   DATA[2664,36] := 1.730048;
   DATA[2664,37] := 188.8618;
   DATA[2664,38] := 0.000128152;
   DATA[2664,39] := 1.0;
   DATA[2664,40] := 1.0;
   DATA[2665,0] := 2.431861;
   DATA[2665,1] := 870.5869;
   DATA[2665,2] := 2.0;
   DATA[2665,3] := 2.0;
   DATA[2665,4] := 262.3366;
   DATA[2665,5] := 8.396757;
   DATA[2665,6] := 329.1464;
   DATA[2665,7] := 2.451799;
   DATA[2665,8] := 2.0;
   DATA[2665,9] := 2.0;
   DATA[2665,10] := 2.0;
   DATA[2665,11] := 19.69396;
   DATA[2665,12] := 2.206322;
   DATA[2665,13] := 834.4415;
   DATA[2665,14] := 1.0;
   DATA[2665,15] := 2.0;
   DATA[2665,16] := 1.0;
   DATA[2665,17] := 1.0;
   DATA[2665,18] := 1.0;
   DATA[2665,19] := 2.0;
   DATA[2665,20] := 148.808;
   DATA[2665,21] := 155.3961;
   DATA[2665,22] := 1.717233;
   DATA[2665,23] := 881.2356;
   DATA[2665,24] := 2.0;
   DATA[2665,25] := 2.0;
   DATA[2665,26] := 7.872853;
   DATA[2665,27] := 144.7065;
   DATA[2665,28] := 261.3432;
   DATA[2665,29] := 12.03538;
   DATA[2665,30] := 1.726352;
   DATA[2665,31] := 1.3119;
   DATA[2665,32] := 0.7352687;
   DATA[2665,33] := 0.3066329;
   DATA[2665,34] := 2.0;
   DATA[2665,35] := 250.0961;
   DATA[2665,36] := 1.730048;
   DATA[2665,37] := 188.8618;
   DATA[2665,38] := 0.000128152;
   DATA[2665,39] := 1.0;
   DATA[2665,40] := 1.0;
   DATA[2666,0] := 2.431861;
   DATA[2666,1] := 870.4692;
   DATA[2666,2] := 2.0;
   DATA[2666,3] := 2.0;
   DATA[2666,4] := 262.3366;
   DATA[2666,5] := 8.396757;
   DATA[2666,6] := 329.1464;
   DATA[2666,7] := 2.451799;
   DATA[2666,8] := 2.0;
   DATA[2666,9] := 2.0;
   DATA[2666,10] := 2.0;
   DATA[2666,11] := 19.72598;
   DATA[2666,12] := 2.206322;
   DATA[2666,13] := 834.4415;
   DATA[2666,14] := 1.0;
   DATA[2666,15] := 2.0;
   DATA[2666,16] := 1.0;
   DATA[2666,17] := 1.0;
   DATA[2666,18] := 1.0;
   DATA[2666,19] := 2.0;
   DATA[2666,20] := 148.808;
   DATA[2666,21] := 155.3961;
   DATA[2666,22] := 1.717233;
   DATA[2666,23] := 881.4663;
   DATA[2666,24] := 2.0;
   DATA[2666,25] := 2.0;
   DATA[2666,26] := 7.872853;
   DATA[2666,27] := 144.7065;
   DATA[2666,28] := 261.3432;
   DATA[2666,29] := 12.03538;
   DATA[2666,30] := 1.726352;
   DATA[2666,31] := 1.30652;
   DATA[2666,32] := 0.7352687;
   DATA[2666,33] := 0.3066329;
   DATA[2666,34] := 2.0;
   DATA[2666,35] := 250.0961;
   DATA[2666,36] := 1.730048;
   DATA[2666,37] := 188.8618;
   DATA[2666,38] := 0.000128152;
   DATA[2666,39] := 1.0;
   DATA[2666,40] := 1.0;
   DATA[2667,0] := 2.455882;
   DATA[2667,1] := 870.5869;
   DATA[2667,2] := 2.0;
   DATA[2667,3] := 2.0;
   DATA[2667,4] := 262.3366;
   DATA[2667,5] := 8.396757;
   DATA[2667,6] := 329.1464;
   DATA[2667,7] := 2.455131;
   DATA[2667,8] := 2.0;
   DATA[2667,9] := 2.0;
   DATA[2667,10] := 2.0;
   DATA[2667,11] := 19.74198;
   DATA[2667,12] := 2.20645;
   DATA[2667,13] := 834.802;
   DATA[2667,14] := 1.0;
   DATA[2667,15] := 2.0;
   DATA[2667,16] := 1.0;
   DATA[2667,17] := 1.0;
   DATA[2667,18] := 1.0;
   DATA[2667,19] := 2.0;
   DATA[2667,20] := 148.808;
   DATA[2667,21] := 155.3961;
   DATA[2667,22] := 1.719156;
   DATA[2667,23] := 882.0431;
   DATA[2667,24] := 2.0;
   DATA[2667,25] := 2.0;
   DATA[2667,26] := 7.872853;
   DATA[2667,27] := 144.7065;
   DATA[2667,28] := 261.3432;
   DATA[2667,29] := 12.03538;
   DATA[2667,30] := 1.726352;
   DATA[2667,31] := 1.311387;
   DATA[2667,32] := 0.7352687;
   DATA[2667,33] := 0.3066329;
   DATA[2667,34] := 2.0;
   DATA[2667,35] := 250.1442;
   DATA[2667,36] := 1.730048;
   DATA[2667,37] := 188.8618;
   DATA[2667,38] := 0.000128152;
   DATA[2667,39] := 1.0;
   DATA[2667,40] := 1.0;
   DATA[2668,0] := 2.50008;
   DATA[2668,1] := 870.3907;
   DATA[2668,2] := 2.0;
   DATA[2668,3] := 2.0;
   DATA[2668,4] := 262.3366;
   DATA[2668,5] := 8.396757;
   DATA[2668,6] := 329.1464;
   DATA[2668,7] := 2.455131;
   DATA[2668,8] := 2.0;
   DATA[2668,9] := 2.0;
   DATA[2668,10] := 2.0;
   DATA[2668,11] := 19.75799;
   DATA[2668,12] := 2.209909;
   DATA[2668,13] := 834.802;
   DATA[2668,14] := 1.0;
   DATA[2668,15] := 2.0;
   DATA[2668,16] := 1.0;
   DATA[2668,17] := 1.0;
   DATA[2668,18] := 1.0;
   DATA[2668,19] := 2.0;
   DATA[2668,20] := 148.808;
   DATA[2668,21] := 155.3961;
   DATA[2668,22] := 1.719156;
   DATA[2668,23] := 882.1969;
   DATA[2668,24] := 2.0;
   DATA[2668,25] := 2.0;
   DATA[2668,26] := 7.872853;
   DATA[2668,27] := 144.7065;
   DATA[2668,28] := 261.3432;
   DATA[2668,29] := 12.03538;
   DATA[2668,30] := 1.726352;
   DATA[2668,31] := 1.313949;
   DATA[2668,32] := 0.7352687;
   DATA[2668,33] := 0.3066329;
   DATA[2668,34] := 2.0;
   DATA[2668,35] := 250.3044;
   DATA[2668,36] := 1.730048;
   DATA[2668,37] := 189.0381;
   DATA[2668,38] := 0.000128152;
   DATA[2668,39] := 1.0;
   DATA[2668,40] := 1.0;
   DATA[2669,0] := 2.537873;
   DATA[2669,1] := 870.7047;
   DATA[2669,2] := 2.0;
   DATA[2669,3] := 2.0;
   DATA[2669,4] := 262.3366;
   DATA[2669,5] := 8.396757;
   DATA[2669,6] := 329.1464;
   DATA[2669,7] := 2.455131;
   DATA[2669,8] := 2.0;
   DATA[2669,9] := 2.0;
   DATA[2669,10] := 2.0;
   DATA[2669,11] := 19.7964;
   DATA[2669,12] := 2.209909;
   DATA[2669,13] := 835.1625;
   DATA[2669,14] := 1.0;
   DATA[2669,15] := 2.0;
   DATA[2669,16] := 1.0;
   DATA[2669,17] := 1.0;
   DATA[2669,18] := 1.0;
   DATA[2669,19] := 2.0;
   DATA[2669,20] := 148.808;
   DATA[2669,21] := 155.3961;
   DATA[2669,22] := 1.719156;
   DATA[2669,23] := 882.2354;
   DATA[2669,24] := 2.0;
   DATA[2669,25] := 2.0;
   DATA[2669,26] := 7.874135;
   DATA[2669,27] := 144.7065;
   DATA[2669,28] := 261.3432;
   DATA[2669,29] := 12.03538;
   DATA[2669,30] := 1.726352;
   DATA[2669,31] := 1.311643;
   DATA[2669,32] := 0.7352687;
   DATA[2669,33] := 0.3066329;
   DATA[2669,34] := 2.0;
   DATA[2669,35] := 250.3044;
   DATA[2669,36] := 1.730048;
   DATA[2669,37] := 189.0541;
   DATA[2669,38] := 0.000128152;
   DATA[2669,39] := 1.0;
   DATA[2669,40] := 1.0;
   DATA[2670,0] := 2.585594;
   DATA[2670,1] := 871.058;
   DATA[2670,2] := 2.0;
   DATA[2670,3] := 2.0;
   DATA[2670,4] := 262.3366;
   DATA[2670,5] := 8.396757;
   DATA[2670,6] := 329.1464;
   DATA[2670,7] := 2.455131;
   DATA[2670,8] := 2.0;
   DATA[2670,9] := 2.0;
   DATA[2670,10] := 2.0;
   DATA[2670,11] := 19.7964;
   DATA[2670,12] := 2.209909;
   DATA[2670,13] := 835.1625;
   DATA[2670,14] := 1.0;
   DATA[2670,15] := 2.0;
   DATA[2670,16] := 1.0;
   DATA[2670,17] := 1.0;
   DATA[2670,18] := 1.0;
   DATA[2670,19] := 2.0;
   DATA[2670,20] := 148.808;
   DATA[2670,21] := 155.3961;
   DATA[2670,22] := 1.717105;
   DATA[2670,23] := 882.3892;
   DATA[2670,24] := 2.0;
   DATA[2670,25] := 2.0;
   DATA[2670,26] := 7.874135;
   DATA[2670,27] := 144.7065;
   DATA[2670,28] := 261.3432;
   DATA[2670,29] := 12.03538;
   DATA[2670,30] := 1.726352;
   DATA[2670,31] := 1.288587;
   DATA[2670,32] := 0.7352687;
   DATA[2670,33] := 0.3066329;
   DATA[2670,34] := 2.0;
   DATA[2670,35] := 250.3044;
   DATA[2670,36] := 1.730048;
   DATA[2670,37] := 189.1182;
   DATA[2670,38] := 0.000128152;
   DATA[2670,39] := 1.0;
   DATA[2670,40] := 1.0;
   DATA[2671,0] := 2.618903;
   DATA[2671,1] := 870.7047;
   DATA[2671,2] := 2.0;
   DATA[2671,3] := 2.0;
   DATA[2671,4] := 262.3366;
   DATA[2671,5] := 8.396757;
   DATA[2671,6] := 329.1464;
   DATA[2671,7] := 2.456156;
   DATA[2671,8] := 2.0;
   DATA[2671,9] := 2.0;
   DATA[2671,10] := 2.0;
   DATA[2671,11] := 19.7804;
   DATA[2671,12] := 2.209909;
   DATA[2671,13] := 835.2025;
   DATA[2671,14] := 1.0;
   DATA[2671,15] := 2.0;
   DATA[2671,16] := 1.0;
   DATA[2671,17] := 1.0;
   DATA[2671,18] := 1.0;
   DATA[2671,19] := 2.0;
   DATA[2671,20] := 148.808;
   DATA[2671,21] := 155.3961;
   DATA[2671,22] := 1.717105;
   DATA[2671,23] := 882.6967;
   DATA[2671,24] := 2.0;
   DATA[2671,25] := 2.0;
   DATA[2671,26] := 7.874135;
   DATA[2671,27] := 144.7065;
   DATA[2671,28] := 261.3432;
   DATA[2671,29] := 12.03538;
   DATA[2671,30] := 1.726352;
   DATA[2671,31] := 1.27296;
   DATA[2671,32] := 0.7352687;
   DATA[2671,33] := 0.3066329;
   DATA[2671,34] := 2.0;
   DATA[2671,35] := 250.3044;
   DATA[2671,36] := 1.730048;
   DATA[2671,37] := 189.1182;
   DATA[2671,38] := 0.000128152;
   DATA[2671,39] := 1.0;
   DATA[2671,40] := 1.0;
   DATA[2672,0] := 2.644845;
   DATA[2672,1] := 871.2542;
   DATA[2672,2] := 2.0;
   DATA[2672,3] := 2.0;
   DATA[2672,4] := 262.3366;
   DATA[2672,5] := 8.396757;
   DATA[2672,6] := 329.1464;
   DATA[2672,7] := 2.456156;
   DATA[2672,8] := 2.0;
   DATA[2672,9] := 2.0;
   DATA[2672,10] := 2.0;
   DATA[2672,11] := 19.73558;
   DATA[2672,12] := 2.209909;
   DATA[2672,13] := 835.2827;
   DATA[2672,14] := 1.0;
   DATA[2672,15] := 2.0;
   DATA[2672,16] := 1.0;
   DATA[2672,17] := 1.0;
   DATA[2672,18] := 1.0;
   DATA[2672,19] := 2.0;
   DATA[2672,20] := 148.808;
   DATA[2672,21] := 155.3961;
   DATA[2672,22] := 1.717105;
   DATA[2672,23] := 882.8121;
   DATA[2672,24] := 2.0;
   DATA[2672,25] := 2.0;
   DATA[2672,26] := 7.874135;
   DATA[2672,27] := 144.7065;
   DATA[2672,28] := 261.3432;
   DATA[2672,29] := 12.03538;
   DATA[2672,30] := 1.726352;
   DATA[2672,31] := 1.265915;
   DATA[2672,32] := 0.7352687;
   DATA[2672,33] := 0.3066329;
   DATA[2672,34] := 2.0;
   DATA[2672,35] := 250.3044;
   DATA[2672,36] := 1.730048;
   DATA[2672,37] := 188.9419;
   DATA[2672,38] := 0.000128152;
   DATA[2672,39] := 1.0;
   DATA[2672,40] := 1.0;
   DATA[2673,0] := 2.658937;
   DATA[2673,1] := 871.058;
   DATA[2673,3] := 2.0;
   DATA[2673,4] := 262.3366;
   DATA[2673,5] := 8.396757;
   DATA[2673,6] := 329.1464;
   DATA[2673,7] := 2.456156;
   DATA[2673,8] := 2.0;
   DATA[2673,9] := 2.0;
   DATA[2673,10] := 2.0;
   DATA[2673,11] := 19.71637;
   DATA[2673,12] := 2.211959;
   DATA[2673,13] := 835.6832;
   DATA[2673,14] := 1.0;
   DATA[2673,15] := 2.0;
   DATA[2673,16] := 1.0;
   DATA[2673,17] := 1.0;
   DATA[2673,18] := 1.0;
   DATA[2673,19] := 2.0;
   DATA[2673,20] := 148.808;
   DATA[2673,21] := 155.3961;
   DATA[2673,22] := 1.717105;
   DATA[2673,23] := 882.6967;
   DATA[2673,24] := 2.0;
   DATA[2673,25] := 2.0;
   DATA[2673,26] := 7.874135;
   DATA[2673,27] := 144.7065;
   DATA[2673,28] := 261.3432;
   DATA[2673,29] := 12.03538;
   DATA[2673,30] := 1.728659;
   DATA[2673,31] := 1.261944;
   DATA[2673,32] := 0.7352687;
   DATA[2673,33] := 0.3066329;
   DATA[2673,34] := 2.0;
   DATA[2673,35] := 250.3044;
   DATA[2673,36] := 1.730048;
   DATA[2673,37] := 188.9419;
   DATA[2673,38] := 0.000128152;
   DATA[2673,39] := 1.0;
   DATA[2673,40] := 1.0;
   DATA[2674,0] := 2.658937;
   DATA[2674,1] := 871.0972;
   DATA[2674,3] := 2.0;
   DATA[2674,4] := 262.3366;
   DATA[2674,5] := 8.396757;
   DATA[2674,6] := 329.1464;
   DATA[2674,7] := 2.453978;
   DATA[2674,8] := 2.0;
   DATA[2674,9] := 2.0;
   DATA[2674,10] := 2.0;
   DATA[2674,11] := 19.71637;
   DATA[2674,12] := 2.212215;
   DATA[2674,13] := 835.563;
   DATA[2674,14] := 1.0;
   DATA[2674,15] := 2.0;
   DATA[2674,16] := 1.0;
   DATA[2674,17] := 1.0;
   DATA[2674,18] := 1.0;
   DATA[2674,19] := 2.0;
   DATA[2674,20] := 148.808;
   DATA[2674,21] := 155.3961;
   DATA[2674,22] := 1.717105;
   DATA[2674,23] := 882.889;
   DATA[2674,24] := 2.0;
   DATA[2674,25] := 2.0;
   DATA[2674,26] := 7.874135;
   DATA[2674,27] := 144.7065;
   DATA[2674,28] := 261.3432;
   DATA[2674,29] := 12.03538;
   DATA[2674,30] := 1.728916;
   DATA[2674,31] := 1.276419;
   DATA[2674,32] := 0.7352687;
   DATA[2674,33] := 0.3066329;
   DATA[2674,34] := 2.0;
   DATA[2674,35] := 250.1442;
   DATA[2674,36] := 1.730048;
   DATA[2674,37] := 188.9419;
   DATA[2674,38] := 0.000128152;
   DATA[2674,39] := 1.0;
   DATA[2674,40] := 1.0;
   DATA[2675,0] := 2.639721;
   DATA[2675,1] := 871.215;
   DATA[2675,3] := 2.0;
   DATA[2675,4] := 262.3366;
   DATA[2675,5] := 8.396757;
   DATA[2675,6] := 329.1464;
   DATA[2675,7] := 2.452952;
   DATA[2675,8] := 2.0;
   DATA[2675,9] := 2.0;
   DATA[2675,10] := 2.0;
   DATA[2675,11] := 19.71637;
   DATA[2675,12] := 2.212215;
   DATA[2675,13] := 835.4028;
   DATA[2675,14] := 1.0;
   DATA[2675,15] := 2.0;
   DATA[2675,16] := 1.0;
   DATA[2675,17] := 1.0;
   DATA[2675,18] := 1.0;
   DATA[2675,19] := 2.0;
   DATA[2675,20] := 148.808;
   DATA[2675,21] := 155.3961;
   DATA[2675,22] := 1.717105;
   DATA[2675,23] := 882.6198;
   DATA[2675,24] := 2.0;
   DATA[2675,25] := 2.0;
   DATA[2675,26] := 7.874135;
   DATA[2675,27] := 144.7065;
   DATA[2675,28] := 261.3432;
   DATA[2675,29] := 11.72776;
   DATA[2675,30] := 1.728916;
   DATA[2675,31] := 1.28167;
   DATA[2675,32] := 0.7352687;
   DATA[2675,33] := 0.3066329;
   DATA[2675,34] := 2.0;
   DATA[2675,35] := 250.1442;
   DATA[2675,36] := 1.730048;
   DATA[2675,37] := 188.9419;
   DATA[2675,38] := 0.000128152;
   DATA[2675,39] := 1.0;
   DATA[2675,40] := 1.0;
   DATA[2676,0] := 2.633635;
   DATA[2676,1] := 870.9794;
   DATA[2676,3] := 2.0;
   DATA[2676,4] := 262.3366;
   DATA[2676,5] := 8.396757;
   DATA[2676,6] := 329.1464;
   DATA[2676,7] := 2.452952;
   DATA[2676,8] := 2.0;
   DATA[2676,9] := 2.0;
   DATA[2676,10] := 2.0;
   DATA[2676,11] := 19.71637;
   DATA[2676,12] := 2.209397;
   DATA[2676,13] := 835.6031;
   DATA[2676,14] := 1.0;
   DATA[2676,15] := 2.0;
   DATA[2676,16] := 1.0;
   DATA[2676,17] := 1.0;
   DATA[2676,18] := 1.0;
   DATA[2676,19] := 2.0;
   DATA[2676,20] := 148.808;
   DATA[2676,21] := 155.5242;
   DATA[2676,22] := 1.717105;
   DATA[2676,23] := 882.5814;
   DATA[2676,24] := 2.0;
   DATA[2676,25] := 2.0;
   DATA[2676,26] := 7.874135;
   DATA[2676,27] := 144.7065;
   DATA[2676,28] := 261.3432;
   DATA[2676,29] := 11.72776;
   DATA[2676,30] := 1.728916;
   DATA[2676,31] := 1.276547;
   DATA[2676,32] := 0.7352687;
   DATA[2676,33] := 0.3066329;
   DATA[2676,34] := 2.0;
   DATA[2676,35] := 250.3525;
   DATA[2676,36] := 1.730048;
   DATA[2676,37] := 189.1182;
   DATA[2676,38] := 0.000128152;
   DATA[2676,39] := 1.0;
   DATA[2676,40] := 1.0;
   DATA[2677,0] := 2.633635;
   DATA[2677,1] := 870.6654;
   DATA[2677,3] := 2.0;
   DATA[2677,4] := 262.3366;
   DATA[2677,5] := 8.396757;
   DATA[2677,6] := 329.1464;
   DATA[2677,7] := 2.452952;
   DATA[2677,8] := 2.0;
   DATA[2677,9] := 2.0;
   DATA[2677,10] := 2.0;
   DATA[2677,11] := 19.71637;
   DATA[2677,12] := 2.209397;
   DATA[2677,13] := 835.4429;
   DATA[2677,14] := 1.0;
   DATA[2677,15] := 2.0;
   DATA[2677,16] := 1.0;
   DATA[2677,17] := 1.0;
   DATA[2677,18] := 1.0;
   DATA[2677,19] := 2.0;
   DATA[2677,20] := 148.808;
   DATA[2677,21] := 155.5242;
   DATA[2677,22] := 1.718515;
   DATA[2677,23] := 882.6967;
   DATA[2677,24] := 2.0;
   DATA[2677,25] := 2.0;
   DATA[2677,26] := 7.874135;
   DATA[2677,27] := 144.7065;
   DATA[2677,28] := 261.3432;
   DATA[2677,29] := 11.72776;
   DATA[2677,30] := 1.730838;
   DATA[2677,31] := 1.280902;
   DATA[2677,32] := 0.7352687;
   DATA[2677,33] := 0.3084905;
   DATA[2677,34] := 2.0;
   DATA[2677,35] := 250.3525;
   DATA[2677,36] := 1.730048;
   DATA[2677,37] := 189.1182;
   DATA[2677,38] := 0.000128152;
   DATA[2677,39] := 1.0;
   DATA[2677,40] := 1.0;
   DATA[2678,0] := 2.625628;
   DATA[2678,1] := 870.6654;
   DATA[2678,3] := 2.0;
   DATA[2678,4] := 262.3366;
   DATA[2678,5] := 8.396757;
   DATA[2678,6] := 329.1464;
   DATA[2678,7] := 2.452952;
   DATA[2678,8] := 2.0;
   DATA[2678,9] := 2.0;
   DATA[2678,10] := 2.0;
   DATA[2678,11] := 19.73878;
   DATA[2678,12] := 2.209397;
   DATA[2678,13] := 835.3627;
   DATA[2678,14] := 1.0;
   DATA[2678,15] := 2.0;
   DATA[2678,16] := 1.0;
   DATA[2678,17] := 1.0;
   DATA[2678,18] := 1.0;
   DATA[2678,19] := 2.0;
   DATA[2678,20] := 148.808;
   DATA[2678,21] := 155.5242;
   DATA[2678,22] := 1.718515;
   DATA[2678,23] := 882.6583;
   DATA[2678,24] := 2.0;
   DATA[2678,25] := 2.0;
   DATA[2678,26] := 7.874135;
   DATA[2678,27] := 144.7065;
   DATA[2678,28] := 261.3432;
   DATA[2678,29] := 12.07383;
   DATA[2678,30] := 1.731735;
   DATA[2678,31] := 1.288203;
   DATA[2678,32] := 0.7352687;
   DATA[2678,33] := 0.3084905;
   DATA[2678,34] := 2.0;
   DATA[2678,35] := 250.4967;
   DATA[2678,36] := 1.730048;
   DATA[2678,37] := 189.2624;
   DATA[2678,38] := 0.000128152;
   DATA[2678,39] := 1.0;
   DATA[2678,40] := 1.0;
   DATA[2679,0] := 2.600006;
   DATA[2679,1] := 871.058;
   DATA[2679,3] := 2.0;
   DATA[2679,4] := 262.3366;
   DATA[2679,5] := 8.396757;
   DATA[2679,6] := 329.1464;
   DATA[2679,7] := 2.452952;
   DATA[2679,8] := 2.0;
   DATA[2679,9] := 2.0;
   DATA[2679,10] := 2.0;
   DATA[2679,11] := 19.74838;
   DATA[2679,12] := 2.209397;
   DATA[2679,13] := 835.0023;
   DATA[2679,14] := 1.0;
   DATA[2679,15] := 2.0;
   DATA[2679,16] := 1.0;
   DATA[2679,17] := 1.0;
   DATA[2679,18] := 1.0;
   DATA[2679,19] := 2.0;
   DATA[2679,20] := 148.808;
   DATA[2679,21] := 155.473;
   DATA[2679,22] := 1.718515;
   DATA[2679,23] := 882.4661;
   DATA[2679,24] := 2.0;
   DATA[2679,25] := 2.0;
   DATA[2679,26] := 7.874135;
   DATA[2679,27] := 144.7065;
   DATA[2679,28] := 261.3432;
   DATA[2679,29] := 12.07383;
   DATA[2679,30] := 1.731735;
   DATA[2679,31] := 1.307416;
   DATA[2679,32] := 0.7352687;
   DATA[2679,33] := 0.3084905;
   DATA[2679,34] := 2.0;
   DATA[2679,35] := 250.4967;
   DATA[2679,36] := 1.730048;
   DATA[2679,37] := 189.2624;
   DATA[2679,38] := 0.000128152;
   DATA[2679,39] := 1.0;
   DATA[2679,40] := 1.0;
   DATA[2680,0] := 2.552285;
   DATA[2680,1] := 870.7047;
   DATA[2680,3] := 2.0;
   DATA[2680,4] := 262.3366;
   DATA[2680,5] := 8.396757;
   DATA[2680,6] := 329.0182;
   DATA[2680,7] := 2.452568;
   DATA[2680,8] := 2.0;
   DATA[2680,9] := 2.0;
   DATA[2680,10] := 2.0;
   DATA[2680,11] := 19.74838;
   DATA[2680,12] := 2.20645;
   DATA[2680,13] := 834.762;
   DATA[2680,14] := 1.0;
   DATA[2680,15] := 2.0;
   DATA[2680,16] := 1.0;
   DATA[2680,17] := 1.0;
   DATA[2680,18] := 1.0;
   DATA[2680,19] := 2.0;
   DATA[2680,20] := 148.808;
   DATA[2680,21] := 155.4473;
   DATA[2680,22] := 1.718515;
   DATA[2680,23] := 882.5045;
   DATA[2680,24] := 2.0;
   DATA[2680,25] := 2.0;
   DATA[2680,26] := 7.870931;
   DATA[2680,27] := 144.7834;
   DATA[2680,28] := 261.3432;
   DATA[2680,29] := 12.07383;
   DATA[2680,30] := 1.731735;
   DATA[2680,31] := 1.320994;
   DATA[2680,32] := 0.7352687;
   DATA[2680,33] := 0.3084905;
   DATA[2680,34] := 2.0;
   DATA[2680,35] := 250.4967;
   DATA[2680,36] := 1.730048;
   DATA[2680,37] := 189.2624;
   DATA[2680,38] := 0.000128152;
   DATA[2680,39] := 1.0;
   DATA[2680,40] := 1.0;
   DATA[2681,0] := 2.499119;
   DATA[2681,1] := 870.8224;
   DATA[2681,3] := 2.0;
   DATA[2681,4] := 262.3366;
   DATA[2681,5] := 8.396757;
   DATA[2681,6] := 329.0182;
   DATA[2681,7] := 2.451671;
   DATA[2681,8] := 2.0;
   DATA[2681,9] := 2.0;
   DATA[2681,10] := 2.0;
   DATA[2681,11] := 19.74838;
   DATA[2681,12] := 2.20645;
   DATA[2681,13] := 834.6818;
   DATA[2681,14] := 1.0;
   DATA[2681,15] := 2.0;
   DATA[2681,16] := 1.0;
   DATA[2681,17] := 1.0;
   DATA[2681,18] := 1.0;
   DATA[2681,19] := 2.0;
   DATA[2681,20] := 148.808;
   DATA[2681,21] := 155.4473;
   DATA[2681,22] := 1.718515;
   DATA[2681,23] := 882.12;
   DATA[2681,24] := 2.0;
   DATA[2681,25] := 2.0;
   DATA[2681,26] := 7.870931;
   DATA[2681,27] := 144.7834;
   DATA[2681,28] := 261.3432;
   DATA[2681,29] := 12.07383;
   DATA[2681,30] := 1.731735;
   DATA[2681,31] := 1.329064;
   DATA[2681,32] := 0.7352687;
   DATA[2681,33] := 0.3084905;
   DATA[2681,34] := 2.0;
   DATA[2681,35] := 250.4967;
   DATA[2681,36] := 1.730048;
   DATA[2681,37] := 189.2624;
   DATA[2681,38] := 0.000128152;
   DATA[2681,39] := 1.0;
   DATA[2681,40] := 1.0;
   DATA[2682,0] := 2.400154;
   DATA[2682,1] := 870.6654;
   DATA[2682,2] := 1.0;
   DATA[2682,3] := 2.0;
   DATA[2682,4] := 262.3366;
   DATA[2682,5] := 8.396757;
   DATA[2682,6] := 329.0182;
   DATA[2682,7] := 2.451671;
   DATA[2682,8] := 2.0;
   DATA[2682,9] := 2.0;
   DATA[2682,10] := 2.0;
   DATA[2682,11] := 19.74838;
   DATA[2682,12] := 2.20645;
   DATA[2682,13] := 835.2025;
   DATA[2682,14] := 1.0;
   DATA[2682,15] := 2.0;
   DATA[2682,16] := 1.0;
   DATA[2682,17] := 1.0;
   DATA[2682,18] := 1.0;
   DATA[2682,19] := 2.0;
   DATA[2682,20] := 148.808;
   DATA[2682,21] := 155.4473;
   DATA[2682,22] := 1.718515;
   DATA[2682,23] := 882.2738;
   DATA[2682,24] := 2.0;
   DATA[2682,25] := 2.0;
   DATA[2682,26] := 7.873815;
   DATA[2682,27] := 144.7834;
   DATA[2682,28] := 261.3432;
   DATA[2682,29] := 12.07383;
   DATA[2682,30] := 1.731351;
   DATA[2682,31] := 1.332138;
   DATA[2682,32] := 0.7352687;
   DATA[2682,33] := 0.3084905;
   DATA[2682,34] := 2.0;
   DATA[2682,35] := 250.4967;
   DATA[2682,36] := 1.730048;
   DATA[2682,37] := 189.2624;
   DATA[2682,38] := 0.000128152;
   DATA[2682,39] := 1.0;
   DATA[2682,40] := 1.0;
   DATA[2683,0] := 2.223361;
   DATA[2683,1] := 870.9794;
   DATA[2683,2] := 1.0;
   DATA[2683,3] := 2.0;
   DATA[2683,4] := 262.3366;
   DATA[2683,5] := 8.396757;
   DATA[2683,6] := 329.0182;
   DATA[2683,7] := 2.451671;
   DATA[2683,8] := 2.0;
   DATA[2683,9] := 2.0;
   DATA[2683,10] := 2.0;
   DATA[2683,11] := 19.74838;
   DATA[2683,12] := 2.20645;
   DATA[2683,13] := 834.6818;
   DATA[2683,14] := 1.0;
   DATA[2683,15] := 2.0;
   DATA[2683,16] := 1.0;
   DATA[2683,17] := 1.0;
   DATA[2683,18] := 1.0;
   DATA[2683,19] := 2.0;
   DATA[2683,20] := 148.808;
   DATA[2683,21] := 155.4473;
   DATA[2683,22] := 1.718515;
   DATA[2683,23] := 882.5045;
   DATA[2683,24] := 2.0;
   DATA[2683,25] := 2.0;
   DATA[2683,26] := 7.874776;
   DATA[2683,27] := 144.7834;
   DATA[2683,28] := 261.3432;
   DATA[2683,29] := 12.07383;
   DATA[2683,30] := 1.731351;
   DATA[2683,31] := 1.31523;
   DATA[2683,32] := 0.7352687;
   DATA[2683,33] := 0.3084905;
   DATA[2683,34] := 2.0;
   DATA[2683,35] := 250.4967;
   DATA[2683,36] := 1.810143;
   DATA[2683,37] := 189.2624;
   DATA[2683,38] := 0.000128152;
   DATA[2683,39] := 1.0;
   DATA[2683,40] := 1.0;
   DATA[2684,0] := 1.916216;
   DATA[2684,1] := 870.5869;
   DATA[2684,2] := 1.0;
   DATA[2684,3] := 2.0;
   DATA[2684,4] := 262.3366;
   DATA[2684,5] := 8.396757;
   DATA[2684,6] := 329.0182;
   DATA[2684,7] := 2.451671;
   DATA[2684,8] := 2.0;
   DATA[2684,9] := 2.0;
   DATA[2684,10] := 2.0;
   DATA[2684,11] := 19.74838;
   DATA[2684,12] := 2.207091;
   DATA[2684,13] := 835.2025;
   DATA[2684,14] := 1.0;
   DATA[2684,15] := 2.0;
   DATA[2684,16] := 1.0;
   DATA[2684,17] := 1.0;
   DATA[2684,18] := 1.0;
   DATA[2684,19] := 2.0;
   DATA[2684,20] := 148.808;
   DATA[2684,21] := 155.3961;
   DATA[2684,22] := 1.716592;
   DATA[2684,23] := 882.5045;
   DATA[2684,24] := 2.0;
   DATA[2684,25] := 2.0;
   DATA[2684,26] := 7.874776;
   DATA[2684,27] := 144.7834;
   DATA[2684,28] := 261.3432;
   DATA[2684,29] := 12.07383;
   DATA[2684,30] := 1.729557;
   DATA[2684,31] := 1.311387;
   DATA[2684,32] := 0.7352687;
   DATA[2684,33] := 0.3084905;
   DATA[2684,34] := 2.0;
   DATA[2684,35] := 250.4967;
   DATA[2684,36] := 1.810143;
   DATA[2684,37] := 189.2624;
   DATA[2684,38] := 0.000128152;
   DATA[2684,39] := 1.0;
   DATA[2684,40] := 1.0;
   DATA[2685,0] := 1.582808;
   DATA[2685,1] := 870.8224;
   DATA[2685,2] := 1.0;
   DATA[2685,3] := 2.0;
   DATA[2685,4] := 262.3366;
   DATA[2685,5] := 8.396757;
   DATA[2685,6] := 329.0182;
   DATA[2685,7] := 2.452952;
   DATA[2685,8] := 2.0;
   DATA[2685,9] := 2.0;
   DATA[2685,10] := 2.0;
   DATA[2685,11] := 19.74838;
   DATA[2685,12] := 2.208756;
   DATA[2685,13] := 834.842;
   DATA[2685,14] := 1.0;
   DATA[2685,15] := 2.0;
   DATA[2685,16] := 1.0;
   DATA[2685,17] := 1.0;
   DATA[2685,18] := 1.0;
   DATA[2685,19] := 2.0;
   DATA[2685,20] := 148.808;
   DATA[2685,21] := 155.3961;
   DATA[2685,22] := 1.716592;
   DATA[2685,23] := 882.2738;
   DATA[2685,24] := 2.0;
   DATA[2685,25] := 2.0;
   DATA[2685,26] := 7.874776;
   DATA[2685,27] := 144.7834;
   DATA[2685,28] := 261.3432;
   DATA[2685,29] := 12.07383;
   DATA[2685,30] := 1.729557;
   DATA[2685,31] := 1.302677;
   DATA[2685,32] := 0.7352687;
   DATA[2685,33] := 0.3066329;
   DATA[2685,34] := 2.0;
   DATA[2685,35] := 250.4967;
   DATA[2685,36] := 1.810143;
   DATA[2685,37] := 189.2624;
   DATA[2685,38] := 0.000128152;
   DATA[2685,39] := 1.0;
   DATA[2685,40] := 1.0;
   DATA[2686,0] := 1.178618;
   DATA[2686,1] := 870.4299;
   DATA[2686,2] := 1.0;
   DATA[2686,3] := 2.0;
   DATA[2686,4] := 262.3366;
   DATA[2686,5] := 8.396757;
   DATA[2686,6] := 329.0182;
   DATA[2686,7] := 2.452952;
   DATA[2686,8] := 2.0;
   DATA[2686,9] := 2.0;
   DATA[2686,10] := 2.0;
   DATA[2686,11] := 19.69076;
   DATA[2686,12] := 2.209525;
   DATA[2686,13] := 835.1625;
   DATA[2686,14] := 1.0;
   DATA[2686,15] := 2.0;
   DATA[2686,16] := 1.0;
   DATA[2686,17] := 1.0;
   DATA[2686,18] := 1.0;
   DATA[2686,19] := 2.0;
   DATA[2686,20] := 148.808;
   DATA[2686,21] := 155.3961;
   DATA[2686,22] := 1.716592;
   DATA[2686,23] := 882.2738;
   DATA[2686,24] := 2.0;
   DATA[2686,25] := 2.0;
   DATA[2686,26] := 7.874776;
   DATA[2686,27] := 144.7834;
   DATA[2686,28] := 261.3432;
   DATA[2686,29] := 11.84312;
   DATA[2686,30] := 1.729557;
   DATA[2686,31] := 1.292814;
   DATA[2686,32] := 0.7352687;
   DATA[2686,33] := 0.3081703;
   DATA[2686,34] := 2.0;
   DATA[2686,35] := 250.4967;
   DATA[2686,36] := 1.730048;
   DATA[2686,37] := 189.2624;
   DATA[2686,38] := 0.000128152;
   DATA[2686,39] := 1.0;
   DATA[2686,40] := 1.0;
   DATA[2687,0] := 0.801012;
   DATA[2687,1] := 870.1944;
   DATA[2687,2] := 1.0;
   DATA[2687,3] := 2.0;
   DATA[2687,4] := 262.3366;
   DATA[2687,5] := 8.396757;
   DATA[2687,6] := 329.0182;
   DATA[2687,7] := 2.452952;
   DATA[2687,8] := 2.0;
   DATA[2687,9] := 2.0;
   DATA[2687,10] := 2.0;
   DATA[2687,11] := 19.69076;
   DATA[2687,12] := 2.209653;
   DATA[2687,13] := 835.0423;
   DATA[2687,14] := 1.0;
   DATA[2687,15] := 2.0;
   DATA[2687,16] := 1.0;
   DATA[2687,17] := 1.0;
   DATA[2687,18] := 1.0;
   DATA[2687,19] := 2.0;
   DATA[2687,20] := 148.808;
   DATA[2687,21] := 155.3961;
   DATA[2687,22] := 1.716592;
   DATA[2687,23] := 882.5814;
   DATA[2687,24] := 2.0;
   DATA[2687,25] := 2.0;
   DATA[2687,26] := 7.874776;
   DATA[2687,27] := 144.7834;
   DATA[2687,28] := 261.3432;
   DATA[2687,29] := 11.84312;
   DATA[2687,30] := 1.729557;
   DATA[2687,31] := 1.27834;
   DATA[2687,32] := 0.7352687;
   DATA[2687,33] := 0.3086827;
   DATA[2687,34] := 2.0;
   DATA[2687,35] := 250.4967;
   DATA[2687,36] := 1.730048;
   DATA[2687,37] := 189.2624;
   DATA[2687,38] := 0.000128152;
   DATA[2687,39] := 1.0;
   DATA[2687,40] := 1.0;
   DATA[2688,0] := 0.4829773;
   DATA[2688,1] := 869.8411;
   DATA[2688,2] := 1.0;
   DATA[2688,3] := 2.0;
   DATA[2688,4] := 262.3366;
   DATA[2688,5] := 8.396757;
   DATA[2688,6] := 329.0182;
   DATA[2688,7] := 2.452952;
   DATA[2688,8] := 2.0;
   DATA[2688,9] := 2.0;
   DATA[2688,10] := 2.0;
   DATA[2688,11] := 19.69076;
   DATA[2688,12] := 2.209653;
   DATA[2688,13] := 835.0423;
   DATA[2688,14] := 1.0;
   DATA[2688,15] := 2.0;
   DATA[2688,16] := 1.0;
   DATA[2688,17] := 1.0;
   DATA[2688,18] := 1.0;
   DATA[2688,19] := 2.0;
   DATA[2688,20] := 148.808;
   DATA[2688,21] := 155.3961;
   DATA[2688,22] := 1.716464;
   DATA[2688,23] := 882.8505;
   DATA[2688,24] := 2.0;
   DATA[2688,25] := 2.0;
   DATA[2688,26] := 7.874776;
   DATA[2688,27] := 144.7834;
   DATA[2688,28] := 261.3432;
   DATA[2688,29] := 11.84312;
   DATA[2688,30] := 1.729557;
   DATA[2688,31] := 1.257589;
   DATA[2688,32] := 0.7352687;
   DATA[2688,33] := 0.3086827;
   DATA[2688,34] := 2.0;
   DATA[2688,35] := 250.4967;
   DATA[2688,36] := 1.730048;
   DATA[2688,37] := 189.2624;
   DATA[2688,38] := 0.000128152;
   DATA[2688,39] := 1.0;
   DATA[2688,40] := 1.0;
   DATA[2689,0] := 0.2844057;
   DATA[2689,1] := 869.8804;
   DATA[2689,2] := 1.0;
   DATA[2689,3] := 2.0;
   DATA[2689,4] := 262.3366;
   DATA[2689,5] := 8.396757;
   DATA[2689,6] := 329.0182;
   DATA[2689,7] := 2.452952;
   DATA[2689,8] := 2.0;
   DATA[2689,9] := 2.0;
   DATA[2689,10] := 2.0;
   DATA[2689,11] := 19.69076;
   DATA[2689,12] := 2.209653;
   DATA[2689,13] := 835.2426;
   DATA[2689,14] := 1.0;
   DATA[2689,15] := 2.0;
   DATA[2689,16] := 1.0;
   DATA[2689,17] := 1.0;
   DATA[2689,18] := 1.0;
   DATA[2689,19] := 2.0;
   DATA[2689,20] := 148.808;
   DATA[2689,21] := 155.3961;
   DATA[2689,22] := 1.716464;
   DATA[2689,23] := 882.7736;
   DATA[2689,24] := 2.0;
   DATA[2689,25] := 2.0;
   DATA[2689,26] := 7.874776;
   DATA[2689,27] := 144.7834;
   DATA[2689,28] := 261.3432;
   DATA[2689,29] := 12.07383;
   DATA[2689,30] := 1.729557;
   DATA[2689,31] := 1.245805;
   DATA[2689,32] := 0.7352687;
   DATA[2689,33] := 0.3086827;
   DATA[2689,34] := 2.0;
   DATA[2689,35] := 250.3525;
   DATA[2689,36] := 1.730048;
   DATA[2689,37] := 189.1342;
   DATA[2689,38] := 0.000128152;
   DATA[2689,39] := 1.0;
   DATA[2689,40] := 1.0;
   DATA[2690,0] := 0.1518112;
   DATA[2690,1] := 869.8019;
   DATA[2690,2] := 1.0;
   DATA[2690,3] := 2.0;
   DATA[2690,4] := 262.3366;
   DATA[2690,5] := 8.396757;
   DATA[2690,6] := 329.0182;
   DATA[2690,7] := 2.452952;
   DATA[2690,8] := 2.0;
   DATA[2690,9] := 2.0;
   DATA[2690,10] := 2.0;
   DATA[2690,11] := 19.70677;
   DATA[2690,12] := 2.209653;
   DATA[2690,13] := 835.2025;
   DATA[2690,14] := 1.0;
   DATA[2690,15] := 2.0;
   DATA[2690,16] := 1.0;
   DATA[2690,17] := 1.0;
   DATA[2690,18] := 1.0;
   DATA[2690,19] := 2.0;
   DATA[2690,20] := 148.808;
   DATA[2690,21] := 155.3961;
   DATA[2690,22] := 1.716464;
   DATA[2690,23] := 882.7736;
   DATA[2690,24] := 2.0;
   DATA[2690,25] := 2.0;
   DATA[2690,26] := 7.874776;
   DATA[2690,27] := 144.7834;
   DATA[2690,28] := 261.3432;
   DATA[2690,29] := 12.22763;
   DATA[2690,30] := 1.731479;
   DATA[2690,31] := 1.244652;
   DATA[2690,32] := 0.7352687;
   DATA[2690,33] := 0.3086827;
   DATA[2690,34] := 2.0;
   DATA[2690,35] := 250.3525;
   DATA[2690,36] := 1.730048;
   DATA[2690,37] := 189.1342;
   DATA[2690,38] := 0.000128152;
   DATA[2690,39] := 1.0;
   DATA[2690,40] := 1.0;
   DATA[2691,0] := 0.07334337;
   DATA[2691,1] := 869.8411;
   DATA[2691,2] := 1.0;
   DATA[2691,3] := 2.0;
   DATA[2691,4] := 262.3366;
   DATA[2691,5] := 8.396757;
   DATA[2691,6] := 329.1207;
   DATA[2691,7] := 2.452952;
   DATA[2691,8] := 2.0;
   DATA[2691,9] := 2.0;
   DATA[2691,10] := 2.0;
   DATA[2691,11] := 19.74198;
   DATA[2691,12] := 2.209653;
   DATA[2691,13] := 835.4429;
   DATA[2691,14] := 1.0;
   DATA[2691,15] := 2.0;
   DATA[2691,16] := 1.0;
   DATA[2691,17] := 1.0;
   DATA[2691,18] := 1.0;
   DATA[2691,19] := 2.0;
   DATA[2691,20] := 148.808;
   DATA[2691,21] := 155.3961;
   DATA[2691,22] := 1.718515;
   DATA[2691,23] := 882.5045;
   DATA[2691,24] := 2.0;
   DATA[2691,25] := 2.0;
   DATA[2691,26] := 7.874776;
   DATA[2691,27] := 144.7834;
   DATA[2691,28] := 261.3432;
   DATA[2691,29] := 12.22763;
   DATA[2691,30] := 1.731479;
   DATA[2691,31] := 1.262713;
   DATA[2691,32] := 0.7352687;
   DATA[2691,33] := 0.3074016;
   DATA[2691,34] := 2.0;
   DATA[2691,35] := 250.2724;
   DATA[2691,36] := 1.730048;
   DATA[2691,37] := 188.958;
   DATA[2691,38] := 0.000128152;
   DATA[2691,39] := 1.0;
   DATA[2691,40] := 1.0;
   DATA[2692,0] := 0.02370048;
   DATA[2692,1] := 869.7234;
   DATA[2692,2] := 1.0;
   DATA[2692,3] := 2.0;
   DATA[2692,4] := 262.3366;
   DATA[2692,5] := 8.396757;
   DATA[2692,6] := 329.1207;
   DATA[2692,7] := 2.452952;
   DATA[2692,8] := 2.0;
   DATA[2692,9] := 2.0;
   DATA[2692,10] := 2.0;
   DATA[2692,11] := 19.74198;
   DATA[2692,12] := 2.209653;
   DATA[2692,13] := 835.4028;
   DATA[2692,14] := 1.0;
   DATA[2692,15] := 2.0;
   DATA[2692,16] := 1.0;
   DATA[2692,17] := 1.0;
   DATA[2692,18] := 1.0;
   DATA[2692,19] := 2.0;
   DATA[2692,20] := 148.808;
   DATA[2692,21] := 155.3961;
   DATA[2692,22] := 1.718515;
   DATA[2692,23] := 882.2738;
   DATA[2692,24] := 2.0;
   DATA[2692,25] := 2.0;
   DATA[2692,26] := 7.874776;
   DATA[2692,27] := 144.7834;
   DATA[2692,28] := 261.3432;
   DATA[2692,29] := 12.22763;
   DATA[2692,30] := 1.729172;
   DATA[2692,31] := 1.271423;
   DATA[2692,32] := 0.7352687;
   DATA[2692,33] := 0.3075937;
   DATA[2692,34] := 2.0;
   DATA[2692,35] := 250.2724;
   DATA[2692,36] := 1.730048;
   DATA[2692,37] := 188.958;
   DATA[2692,38] := 0.000128152;
   DATA[2692,39] := 1.0;
   DATA[2692,40] := 1.0;
   DATA[2693,0] := 0.000640553;
   DATA[2693,1] := 869.7234;
   DATA[2693,2] := 1.0;
   DATA[2693,3] := 2.0;
   DATA[2693,4] := 262.3366;
   DATA[2693,5] := 8.396757;
   DATA[2693,6] := 329.1464;
   DATA[2693,7] := 2.452952;
   DATA[2693,8] := 2.0;
   DATA[2693,9] := 2.0;
   DATA[2693,10] := 2.0;
   DATA[2693,11] := 19.74198;
   DATA[2693,12] := 2.207091;
   DATA[2693,13] := 835.8033;
   DATA[2693,14] := 1.0;
   DATA[2693,15] := 2.0;
   DATA[2693,16] := 1.0;
   DATA[2693,17] := 1.0;
   DATA[2693,18] := 1.0;
   DATA[2693,19] := 2.0;
   DATA[2693,20] := 148.808;
   DATA[2693,21] := 155.3961;
   DATA[2693,22] := 1.718515;
   DATA[2693,23] := 882.8121;
   DATA[2693,24] := 2.0;
   DATA[2693,25] := 2.0;
   DATA[2693,26] := 7.874776;
   DATA[2693,27] := 144.7834;
   DATA[2693,28] := 261.3432;
   DATA[2693,29] := 12.22763;
   DATA[2693,30] := 1.729172;
   DATA[2693,31] := 1.272064;
   DATA[2693,32] := 0.7352687;
   DATA[2693,33] := 0.3082983;
   DATA[2693,34] := 2.0;
   DATA[2693,35] := 250.2724;
   DATA[2693,36] := 1.730048;
   DATA[2693,37] := 188.958;
   DATA[2693,38] := 0.000128152;
   DATA[2693,39] := 1.0;
   DATA[2693,40] := 1.0;

END_DATA_BLOCK

DATA_BLOCK "DB_FeatureNormRef_std"
{ S7_Optimized_Access := 'TRUE' }
VERSION : 0.1
NON_RETAIN
   VAR
      std : Array[0..39] of Real;
   END_VAR


BEGIN
   std[0] := 1.134874;
   std[1] := 131.2155;
   std[2] := 0.4579044;
   std[3] := 0.436374;
   std[4] := 5.261742;
   std[5] := 0.1128395;
   std[6] := 59.83524;
   std[7] := 1.067913;
   std[8] := 0.4456327;
   std[9] := 0.4373973;
   std[10] := 0.4899075;
   std[11] := 6.801564;
   std[12] := 0.8329131;
   std[13] := 117.8872;
   std[14] := 0.1100685;
   std[15] := 0.419305;
   std[16] := 0.1684625;
   std[17] := 0.1948795;
   std[18] := 0.08104688;
   std[19] := 0.3893126;
   std[20] := 66.43026;
   std[21] := 11.66761;
   std[22] := 0.1758617;
   std[23] := 113.9631;
   std[24] := 0.1028308;
   std[25] := 0.1029105;
   std[26] := 0.06156169;
   std[27] := 11.32486;
   std[28] := 5.737159;
   std[29] := 11.95808;
   std[30] := 0.1767241;
   std[31] := 0.1317653;
   std[32] := 0.0767542;
   std[33] := 0.03271202;
   std[34] := 0.105228;
   std[35] := 25.34136;
   std[36] := 0.2577594;
   std[37] := 19.61726;
   std[38] := 0.1478796;
   std[39] := 0.08817827;

END_DATA_BLOCK

DATA_BLOCK "DB_FeatureNormRef_Means"
{ S7_Optimized_Access := 'TRUE' }
VERSION : 0.1
NON_RETAIN
   VAR
      Means : Array[0..39] of Real;
   END_VAR


BEGIN
   Means[0] := 1.846544;
   Means[1] := 582.3317;
   Means[2] := 1.719179;
   Means[3] := 1.744085;
   Means[4] := 262.3805;
   Means[5] := 8.393863;
   Means[6] := 361.9682;
   Means[7] := 1.824498;
   Means[8] := 1.741861;
   Means[9] := 1.742247;
   Means[10] := 1.599953;
   Means[11] := 16.52142;
   Means[12] := 1.820565;
   Means[13] := 891.7278;
   Means[14] := 1.005415;
   Means[15] := 1.795682;
   Means[16] := 1.019948;
   Means[17] := 1.024403;
   Means[18] := 1.006612;
   Means[19] := 1.813745;
   Means[20] := 107.9063;
   Means[21] := 178.6221;
   Means[22] := 1.683628;
   Means[23] := 872.4719;
   Means[24] := 1.989312;
   Means[25] := 1.989295;
   Means[26] := 7.859592;
   Means[27] := 167.5583;
   Means[28] := 265.8126;
   Means[29] := 12.47605;
   Means[30] := 1.693144;
   Means[31] := 1.252732;
   Means[32] := 0.7332894;
   Means[33] := 0.3058438;
   Means[34] := 1.988802;
   Means[35] := 251.657;
   Means[36] := 1.217715;
   Means[37] := 191.1807;
   Means[38] := 0.0142492;
   Means[39] := 1.007837;

END_DATA_BLOCK

DATA_BLOCK "DB_model_HS16_IW10"
{ S7_Optimized_Access := 'TRUE' }
VERSION : 0.1
NON_RETAIN
// --- Siemens Structured Format ---
   VAR
      W_i : Array[0..15, 0..39] of Real;
      W_f : Array[0..15, 0..39] of Real;
      W_g : Array[0..15, 0..39] of Real;
      W_o : Array[0..15, 0..39] of Real;
      R_i : Array[0..15, 0..15] of Real;
      R_f : Array[0..15, 0..15] of Real;
      R_g : Array[0..15, 0..15] of Real;
      R_o : Array[0..15, 0..15] of Real;
      B_i : Array[0..15] of Real;
      B_f : Array[0..15] of Real;
      B_g : Array[0..15] of Real;
      B_o : Array[0..15] of Real;
      FC_W : Array[0..39, 0..15] of Real;
      FC_B : Array[0..39] of Real;
   END_VAR


BEGIN
   W_i[0,0] := 0.03254747;
   W_i[0,1] := 0.123859;
   W_i[0,2] := 0.04015401;
   W_i[0,3] := -0.03803189;
   W_i[0,4] := 0.1759319;
   W_i[0,5] := 0.00417833;
   W_i[0,6] := -0.00157293;
   W_i[0,7] := 0.0728622;
   W_i[0,8] := 0.06175515;
   W_i[0,9] := -0.03080547;
   W_i[0,10] := 0.01361996;
   W_i[0,11] := -0.2367004;
   W_i[0,12] := 0.1251248;
   W_i[0,13] := -0.1203895;
   W_i[0,14] := 0.0523482;
   W_i[0,15] := 0.2630532;
   W_i[0,16] := -0.1147504;
   W_i[0,17] := 0.05957858;
   W_i[0,18] := -0.02271187;
   W_i[0,19] := -0.04982074;
   W_i[0,20] := 0.01270425;
   W_i[0,21] := 0.3620531;
   W_i[0,22] := -0.2914467;
   W_i[0,23] := 0.02366253;
   W_i[0,24] := -0.602429;
   W_i[0,25] := -0.5198534;
   W_i[0,26] := 0.01890776;
   W_i[0,27] := -0.4244256;
   W_i[0,28] := 0.09802054;
   W_i[0,29] := -0.2919731;
   W_i[0,30] := 0.1756448;
   W_i[0,31] := -0.06584074;
   W_i[0,32] := 0.04272554;
   W_i[0,33] := 0.06813997;
   W_i[0,34] := 0.1243908;
   W_i[0,35] := -0.2062567;
   W_i[0,36] := 0.05875245;
   W_i[0,37] := -0.2700093;
   W_i[0,38] := 0.2212317;
   W_i[0,39] := 1.454268;
   W_i[1,0] := 0.04402059;
   W_i[1,1] := 0.1007617;
   W_i[1,2] := -0.00997876;
   W_i[1,3] := 0.00796912;
   W_i[1,4] := -0.00383734;
   W_i[1,5] := -0.00800767;
   W_i[1,6] := 0.1229124;
   W_i[1,7] := 0.04417216;
   W_i[1,8] := -0.00160155;
   W_i[1,9] := -0.03973384;
   W_i[1,10] := -0.05576275;
   W_i[1,11] := 0.01415846;
   W_i[1,12] := -0.1102211;
   W_i[1,13] := 0.0361371;
   W_i[1,14] := -0.00464776;
   W_i[1,15] := -0.02071899;
   W_i[1,16] := 0.0165178;
   W_i[1,17] := -0.00011115;
   W_i[1,18] := 0.04986879;
   W_i[1,19] := -0.05042609;
   W_i[1,20] := 0.08610544;
   W_i[1,21] := 0.05673008;
   W_i[1,22] := -0.00434864;
   W_i[1,23] := 0.01197722;
   W_i[1,24] := -0.5458539;
   W_i[1,25] := -0.6899631;
   W_i[1,26] := 0.01104975;
   W_i[1,27] := 0.0182511;
   W_i[1,28] := 0.04478757;
   W_i[1,29] := -0.05586376;
   W_i[1,30] := 0.02979602;
   W_i[1,31] := 0.00707946;
   W_i[1,32] := 0.1464935;
   W_i[1,33] := 0.04832766;
   W_i[1,34] := -0.9202742;
   W_i[1,35] := -0.1918912;
   W_i[1,36] := 0.02485085;
   W_i[1,37] := -0.05241579;
   W_i[1,38] := 0.01553158;
   W_i[1,39] := -0.00394726;
   W_i[2,0] := 0.0670436;
   W_i[2,1] := -0.1175203;
   W_i[2,2] := 0.02326228;
   W_i[2,3] := -0.1431773;
   W_i[2,4] := -0.05582308;
   W_i[2,5] := 0.03605313;
   W_i[2,6] := 0.04952687;
   W_i[2,7] := -0.05419854;
   W_i[2,8] := -0.00077774;
   W_i[2,9] := 0.1769989;
   W_i[2,10] := 0.02469403;
   W_i[2,11] := 0.2849406;
   W_i[2,12] := -0.2712711;
   W_i[2,13] := -0.06837726;
   W_i[2,14] := 0.00509281;
   W_i[2,15] := 0.07467768;
   W_i[2,16] := 0.01470727;
   W_i[2,17] := 0.1139419;
   W_i[2,18] := -0.03895494;
   W_i[2,19] := 0.02999579;
   W_i[2,20] := 0.0196714;
   W_i[2,21] := 0.00220801;
   W_i[2,22] := -0.33803;
   W_i[2,23] := 0.09799825;
   W_i[2,24] := -0.5955718;
   W_i[2,25] := -0.7228485;
   W_i[2,26] := 0.07928592;
   W_i[2,27] := -0.03053538;
   W_i[2,28] := -0.1309938;
   W_i[2,29] := -0.04490006;
   W_i[2,30] := 0.05262627;
   W_i[2,31] := -0.03356259;
   W_i[2,32] := 0.06378829;
   W_i[2,33] := -0.00362085;
   W_i[2,34] := -0.6579466;
   W_i[2,35] := 0.02030313;
   W_i[2,36] := 0.05807094;
   W_i[2,37] := -0.1117615;
   W_i[2,38] := 0.09806133;
   W_i[2,39] := -0.04513157;
   W_i[3,0] := -0.03288125;
   W_i[3,1] := 0.03644303;
   W_i[3,2] := -0.02111984;
   W_i[3,3] := -0.09554495;
   W_i[3,4] := 0.471034;
   W_i[3,5] := -0.0182176;
   W_i[3,6] := -0.01296977;
   W_i[3,7] := 0.09772011;
   W_i[3,8] := 0.02375359;
   W_i[3,9] := 0.0802948;
   W_i[3,10] := 0.06341432;
   W_i[3,11] := -0.05777879;
   W_i[3,12] := 0.09200994;
   W_i[3,13] := -0.0054342;
   W_i[3,14] := -0.1107964;
   W_i[3,15] := 0.1856784;
   W_i[3,16] := -0.0179559;
   W_i[3,17] := -0.01424691;
   W_i[3,18] := 0.02418556;
   W_i[3,19] := -0.08783326;
   W_i[3,20] := 0.05560731;
   W_i[3,21] := 0.2986822;
   W_i[3,22] := -0.2220259;
   W_i[3,23] := -0.03734203;
   W_i[3,24] := 0.08825689;
   W_i[3,25] := 0.1838893;
   W_i[3,26] := 0.1152585;
   W_i[3,27] := -0.444976;
   W_i[3,28] := 0.1019801;
   W_i[3,29] := -0.4402614;
   W_i[3,30] := -0.2070405;
   W_i[3,31] := 0.00454621;
   W_i[3,32] := -0.03864358;
   W_i[3,33] := -0.1032195;
   W_i[3,34] := 0.6178231;
   W_i[3,35] := -0.01621445;
   W_i[3,36] := 0.06078746;
   W_i[3,37] := 0.07829241;
   W_i[3,38] := 0.08872399;
   W_i[3,39] := 0.01815886;
   W_i[4,0] := -0.09336383;
   W_i[4,1] := 0.00870158;
   W_i[4,2] := -0.0504511;
   W_i[4,3] := 0.0685437;
   W_i[4,4] := 0.06657482;
   W_i[4,5] := -0.04358229;
   W_i[4,6] := 0.01173393;
   W_i[4,7] := 0.02832152;
   W_i[4,8] := -0.2380867;
   W_i[4,9] := 0.2590344;
   W_i[4,10] := -0.02959821;
   W_i[4,11] := -0.1970284;
   W_i[4,12] := -0.04782372;
   W_i[4,13] := 0.00693473;
   W_i[4,14] := 0.00193878;
   W_i[4,15] := 0.03396931;
   W_i[4,16] := -0.03933699;
   W_i[4,17] := -0.09345319;
   W_i[4,18] := 0.8571873;
   W_i[4,19] := -0.208394;
   W_i[4,20] := -0.00447866;
   W_i[4,21] := -0.04350503;
   W_i[4,22] := 0.09176219;
   W_i[4,23] := 0.04992297;
   W_i[4,24] := -0.4504299;
   W_i[4,25] := 0.01641427;
   W_i[4,26] := -0.1837832;
   W_i[4,27] := 0.03955682;
   W_i[4,28] := -0.06913128;
   W_i[4,29] := 0.08025265;
   W_i[4,30] := -0.1162292;
   W_i[4,31] := 0.04558431;
   W_i[4,32] := 0.07176397;
   W_i[4,33] := -0.04032118;
   W_i[4,34] := 0.2098121;
   W_i[4,35] := -0.1125335;
   W_i[4,36] := -0.01868857;
   W_i[4,37] := -0.07242457;
   W_i[4,38] := -0.1324239;
   W_i[4,39] := -0.04244877;
   W_i[5,0] := 0.01391891;
   W_i[5,1] := -0.110183;
   W_i[5,2] := -0.00893384;
   W_i[5,3] := -0.01407803;
   W_i[5,4] := 0.08575681;
   W_i[5,5] := 0.08241521;
   W_i[5,6] := -0.06153676;
   W_i[5,7] := 0.03060099;
   W_i[5,8] := -0.03490681;
   W_i[5,9] := 0.0314279;
   W_i[5,10] := -0.02459875;
   W_i[5,11] := 0.1095907;
   W_i[5,12] := -0.02965787;
   W_i[5,13] := 0.00184801;
   W_i[5,14] := 0.02055808;
   W_i[5,15] := -0.00937524;
   W_i[5,16] := -0.01257727;
   W_i[5,17] := 0.01791891;
   W_i[5,18] := -0.0115625;
   W_i[5,19] := -0.02731706;
   W_i[5,20] := 0.08900256;
   W_i[5,21] := 0.09895428;
   W_i[5,22] := 0.02720478;
   W_i[5,23] := 0.04369688;
   W_i[5,24] := -1.906074;
   W_i[5,25] := -0.09418426;
   W_i[5,26] := -0.010597;
   W_i[5,27] := -0.09780212;
   W_i[5,28] := 0.1125583;
   W_i[5,29] := 0.08197493;
   W_i[5,30] := -0.08072126;
   W_i[5,31] := 0.03083795;
   W_i[5,32] := 0.06895962;
   W_i[5,33] := 0.00149198;
   W_i[5,34] := 0.3009818;
   W_i[5,35] := 0.1442458;
   W_i[5,36] := -0.02817895;
   W_i[5,37] := -0.08498497;
   W_i[5,38] := 0.03758771;
   W_i[5,39] := 0.01095005;
   W_i[6,0] := 0.08324189;
   W_i[6,1] := -0.2883669;
   W_i[6,2] := -0.00092833;
   W_i[6,3] := -0.00874277;
   W_i[6,4] := 0.1196982;
   W_i[6,5] := -0.1120785;
   W_i[6,6] := -0.0087709;
   W_i[6,7] := -0.03745995;
   W_i[6,8] := 0.00287988;
   W_i[6,9] := 0.00178848;
   W_i[6,10] := 0.03823818;
   W_i[6,11] := 0.02621512;
   W_i[6,12] := -0.288421;
   W_i[6,13] := -0.07084718;
   W_i[6,14] := 0.04070705;
   W_i[6,15] := -0.020424;
   W_i[6,16] := -0.00164282;
   W_i[6,17] := 0.01065832;
   W_i[6,18] := 0.00655926;
   W_i[6,19] := 0.02358968;
   W_i[6,20] := 0.1303789;
   W_i[6,21] := 0.038681;
   W_i[6,22] := -0.06235948;
   W_i[6,23] := 0.07983913;
   W_i[6,24] := -0.2428008;
   W_i[6,25] := -0.05732525;
   W_i[6,26] := 0.1651715;
   W_i[6,27] := -0.07414961;
   W_i[6,28] := 0.06032364;
   W_i[6,29] := 0.08282514;
   W_i[6,30] := -0.01358633;
   W_i[6,31] := 0.0431109;
   W_i[6,32] := 0.03472897;
   W_i[6,33] := -0.04253995;
   W_i[6,34] := 0.01447233;
   W_i[6,35] := 0.03594886;
   W_i[6,36] := -0.01385077;
   W_i[6,37] := 0.1116451;
   W_i[6,38] := 0.1253235;
   W_i[6,39] := -0.03726343;
   W_i[7,0] := 0.01927893;
   W_i[7,1] := 0.05625859;
   W_i[7,2] := 0.04672581;
   W_i[7,3] := -0.00316564;
   W_i[7,4] := 0.09401099;
   W_i[7,5] := -0.02755413;
   W_i[7,6] := -0.03952036;
   W_i[7,7] := 0.03364034;
   W_i[7,8] := 0.05500693;
   W_i[7,9] := 0.02471298;
   W_i[7,10] := 0.03820876;
   W_i[7,11] := -0.2692161;
   W_i[7,12] := -0.02231521;
   W_i[7,13] := -0.0175243;
   W_i[7,14] := 0.03934914;
   W_i[7,15] := 0.01282423;
   W_i[7,16] := -0.0871601;
   W_i[7,17] := -0.09125534;
   W_i[7,18] := 0.00613662;
   W_i[7,19] := 0.08651425;
   W_i[7,20] := -0.01288831;
   W_i[7,21] := 0.2017677;
   W_i[7,22] := -0.2016672;
   W_i[7,23] := 0.01241351;
   W_i[7,24] := -0.8755623;
   W_i[7,25] := -0.4621839;
   W_i[7,26] := 0.09773878;
   W_i[7,27] := -0.1281056;
   W_i[7,28] := 0.04194518;
   W_i[7,29] := -0.03563948;
   W_i[7,30] := 0.08049577;
   W_i[7,31] := 0.04509509;
   W_i[7,32] := -0.113328;
   W_i[7,33] := 0.1053996;
   W_i[7,34] := 0.2416716;
   W_i[7,35] := 0.04508473;
   W_i[7,36] := 0.00324964;
   W_i[7,37] := 0.2255004;
   W_i[7,38] := 0.1750992;
   W_i[7,39] := -0.7787634;
   W_i[8,0] := -0.03076644;
   W_i[8,1] := 0.03958185;
   W_i[8,2] := 0.05958826;
   W_i[8,3] := 0.00143461;
   W_i[8,4] := -0.03551066;
   W_i[8,5] := 0.0670559;
   W_i[8,6] := -0.00545013;
   W_i[8,7] := -0.1152002;
   W_i[8,8] := -0.04941865;
   W_i[8,9] := 0.00970779;
   W_i[8,10] := -0.02700928;
   W_i[8,11] := 0.1261697;
   W_i[8,12] := -0.230127;
   W_i[8,13] := -0.1321811;
   W_i[8,14] := 0.1056539;
   W_i[8,15] := 0.03265957;
   W_i[8,16] := 0.01893855;
   W_i[8,17] := 0.05783269;
   W_i[8,18] := 0.04541522;
   W_i[8,19] := -0.1756509;
   W_i[8,20] := -0.0300831;
   W_i[8,21] := 0.02609591;
   W_i[8,22] := -0.1179207;
   W_i[8,23] := -0.03097328;
   W_i[8,24] := -1.123494;
   W_i[8,25] := -0.1057856;
   W_i[8,26] := 0.1196709;
   W_i[8,27] := -0.1930985;
   W_i[8,28] := -0.04314341;
   W_i[8,29] := -0.02280886;
   W_i[8,30] := 0.09419166;
   W_i[8,31] := -0.00168002;
   W_i[8,32] := 0.170113;
   W_i[8,33] := 0.1277638;
   W_i[8,34] := 0.0079219;
   W_i[8,35] := 0.00793266;
   W_i[8,36] := 0.02933485;
   W_i[8,37] := -0.04765635;
   W_i[8,38] := -0.05385318;
   W_i[8,39] := 1.045761;
   W_i[9,0] := 0.1591891;
   W_i[9,1] := 0.04106269;
   W_i[9,2] := 0.02940365;
   W_i[9,3] := -0.02633034;
   W_i[9,4] := 0.06646424;
   W_i[9,5] := -0.06870057;
   W_i[9,6] := 0.00617184;
   W_i[9,7] := 0.01493581;
   W_i[9,8] := 0.00472299;
   W_i[9,9] := -0.1817109;
   W_i[9,10] := -0.0086358;
   W_i[9,11] := 0.1120397;
   W_i[9,12] := 0.03235663;
   W_i[9,13] := -0.00635904;
   W_i[9,14] := -0.00805719;
   W_i[9,15] := 0.03256573;
   W_i[9,16] := -0.029828;
   W_i[9,17] := 0.02432551;
   W_i[9,18] := -0.04791717;
   W_i[9,19] := -0.03479305;
   W_i[9,20] := 0.02419964;
   W_i[9,21] := -0.0080657;
   W_i[9,22] := 0.00884045;
   W_i[9,23] := 0.00822151;
   W_i[9,24] := -0.4626606;
   W_i[9,25] := -0.2415425;
   W_i[9,26] := 0.1063772;
   W_i[9,27] := 0.00555547;
   W_i[9,28] := 0.00231378;
   W_i[9,29] := 0.1730648;
   W_i[9,30] := -0.1442872;
   W_i[9,31] := -0.01611738;
   W_i[9,32] := -0.1527355;
   W_i[9,33] := -0.03995335;
   W_i[9,34] := -0.6023377;
   W_i[9,35] := -0.06071381;
   W_i[9,36] := 0.01153921;
   W_i[9,37] := 0.157252;
   W_i[9,38] := 0.04887648;
   W_i[9,39] := 0.03194974;
   W_i[10,0] := 5.71E-06;
   W_i[10,1] := 0.0292189;
   W_i[10,2] := 0.03921259;
   W_i[10,3] := -0.1034236;
   W_i[10,4] := 0.04451175;
   W_i[10,5] := -0.01788418;
   W_i[10,6] := 0.06014212;
   W_i[10,7] := -0.127616;
   W_i[10,8] := 0.1096968;
   W_i[10,9] := 0.1346427;
   W_i[10,10] := -0.07629871;
   W_i[10,11] := -1.314735;
   W_i[10,12] := 0.9704102;
   W_i[10,13] := -0.02917644;
   W_i[10,14] := 0.2685799;
   W_i[10,15] := 0.06801854;
   W_i[10,16] := -0.2241947;
   W_i[10,17] := 0.2624845;
   W_i[10,18] := -0.1694944;
   W_i[10,19] := -0.1197102;
   W_i[10,20] := -0.1591434;
   W_i[10,21] := 0.1818019;
   W_i[10,22] := -0.4487775;
   W_i[10,23] := 0.05718501;
   W_i[10,24] := 0.7740152;
   W_i[10,25] := 0.6112806;
   W_i[10,26] := 0.00735129;
   W_i[10,27] := -0.08243502;
   W_i[10,28] := -0.03729297;
   W_i[10,29] := 0.1612841;
   W_i[10,30] := -0.02351914;
   W_i[10,31] := 0.1043125;
   W_i[10,32] := 0.05746254;
   W_i[10,33] := 0.08887602;
   W_i[10,34] := -0.3910645;
   W_i[10,35] := 0.2256924;
   W_i[10,36] := -0.1320819;
   W_i[10,37] := -0.1611588;
   W_i[10,38] := 0.2708046;
   W_i[10,39] := 0.6280136;
   W_i[11,0] := -0.05849513;
   W_i[11,1] := -0.03062119;
   W_i[11,2] := -0.00411083;
   W_i[11,3] := 0.00799791;
   W_i[11,4] := 0.08333463;
   W_i[11,5] := 0.02937987;
   W_i[11,6] := 0.06844535;
   W_i[11,7] := -0.0119828;
   W_i[11,8] := 0.05660131;
   W_i[11,9] := -0.1460933;
   W_i[11,10] := -0.01666861;
   W_i[11,11] := -0.06908122;
   W_i[11,12] := 0.1548331;
   W_i[11,13] := -0.00687739;
   W_i[11,14] := 0.01971146;
   W_i[11,15] := 0.1330592;
   W_i[11,16] := -0.02189317;
   W_i[11,17] := 0.00985993;
   W_i[11,18] := -0.1488067;
   W_i[11,19] := 0.01909257;
   W_i[11,20] := 0.03714932;
   W_i[11,21] := -0.02673176;
   W_i[11,22] := -0.02788893;
   W_i[11,23] := 0.1140895;
   W_i[11,24] := -0.3711884;
   W_i[11,25] := -0.08985706;
   W_i[11,26] := -0.1102327;
   W_i[11,27] := 0.05117378;
   W_i[11,28] := 0.08547711;
   W_i[11,29] := 0.1270248;
   W_i[11,30] := 0.1054488;
   W_i[11,31] := -0.00480978;
   W_i[11,32] := 0.1614495;
   W_i[11,33] := 0.05210381;
   W_i[11,34] := -0.00085451;
   W_i[11,35] := -0.00874526;
   W_i[11,36] := -0.0616112;
   W_i[11,37] := -0.3677483;
   W_i[11,38] := 0.04212995;
   W_i[11,39] := 0.03037546;
   W_i[12,0] := 0.00629061;
   W_i[12,1] := -0.06136212;
   W_i[12,2] := -0.00718669;
   W_i[12,3] := -0.1004218;
   W_i[12,4] := 0.06293897;
   W_i[12,5] := -0.03143417;
   W_i[12,6] := -0.03538829;
   W_i[12,7] := 0.07763195;
   W_i[12,8] := -0.01023159;
   W_i[12,9] := -0.1141296;
   W_i[12,10] := -0.01354402;
   W_i[12,11] := -0.02311977;
   W_i[12,12] := 0.0279608;
   W_i[12,13] := 0.07165248;
   W_i[12,14] := -0.03632027;
   W_i[12,15] := 0.03878558;
   W_i[12,16] := -0.073125;
   W_i[12,17] := 0.01845204;
   W_i[12,18] := -0.08527449;
   W_i[12,19] := -0.00854577;
   W_i[12,20] := 0.00351815;
   W_i[12,21] := -0.1662848;
   W_i[12,22] := 0.06705266;
   W_i[12,23] := 0.1430702;
   W_i[12,24] := -0.539574;
   W_i[12,25] := -0.8721982;
   W_i[12,26] := -0.06440469;
   W_i[12,27] := 0.07379381;
   W_i[12,28] := 0.07828815;
   W_i[12,29] := 0.3882209;
   W_i[12,30] := 0.1159498;
   W_i[12,31] := 0.05581488;
   W_i[12,32] := 0.3066402;
   W_i[12,33] := 0.1275958;
   W_i[12,34] := -0.147978;
   W_i[12,35] := 0.1432935;
   W_i[12,36] := 0.2298153;
   W_i[12,37] := 0.00895516;
   W_i[12,38] := 0.2001298;
   W_i[12,39] := 0.09707437;
   W_i[13,0] := 0.07871004;
   W_i[13,1] := 0.0640982;
   W_i[13,2] := -0.00181766;
   W_i[13,3] := 0.05780525;
   W_i[13,4] := 0.2101672;
   W_i[13,5] := 0.05360549;
   W_i[13,6] := -0.0875827;
   W_i[13,7] := -0.3342811;
   W_i[13,8] := -0.09135646;
   W_i[13,9] := 0.1170631;
   W_i[13,10] := -0.0523126;
   W_i[13,11] := -0.03317479;
   W_i[13,12] := -0.403383;
   W_i[13,13] := -0.00985299;
   W_i[13,14] := 0.02202887;
   W_i[13,15] := 0.130378;
   W_i[13,16] := 0.04808246;
   W_i[13,17] := 0.04501719;
   W_i[13,18] := -0.01153503;
   W_i[13,19] := 0.03141625;
   W_i[13,20] := 0.02999944;
   W_i[13,21] := 0.01402024;
   W_i[13,22] := 0.06788336;
   W_i[13,23] := -0.09942459;
   W_i[13,24] := 0.3184399;
   W_i[13,25] := 0.1069793;
   W_i[13,26] := -0.06989229;
   W_i[13,27] := 0.1058815;
   W_i[13,28] := 0.06872193;
   W_i[13,29] := -0.1537144;
   W_i[13,30] := 0.06626805;
   W_i[13,31] := -0.0559484;
   W_i[13,32] := -0.09573574;
   W_i[13,33] := 0.05669653;
   W_i[13,34] := 0.06202357;
   W_i[13,35] := -0.1367418;
   W_i[13,36] := 0.06451428;
   W_i[13,37] := 0.1204168;
   W_i[13,38] := -0.168509;
   W_i[13,39] := 0.9775926;
   W_i[14,0] := 0.00773311;
   W_i[14,1] := -0.06673568;
   W_i[14,2] := -0.03463669;
   W_i[14,3] := -0.07830913;
   W_i[14,4] := 0.22799;
   W_i[14,5] := -0.2344869;
   W_i[14,6] := 0.1956936;
   W_i[14,7] := 0.1315334;
   W_i[14,8] := -0.1242086;
   W_i[14,9] := 0.2860397;
   W_i[14,10] := -0.09231006;
   W_i[14,11] := -0.2547791;
   W_i[14,12] := 0.1490363;
   W_i[14,13] := -0.2912802;
   W_i[14,14] := 0.1072571;
   W_i[14,15] := 0.1354038;
   W_i[14,16] := -0.09035023;
   W_i[14,17] := -0.01749873;
   W_i[14,18] := -0.4789497;
   W_i[14,19] := -0.06870104;
   W_i[14,20] := -0.1709639;
   W_i[14,21] := -0.05212005;
   W_i[14,22] := -0.1618474;
   W_i[14,23] := -0.2139406;
   W_i[14,24] := -0.7570689;
   W_i[14,25] := -0.7048593;
   W_i[14,26] := -0.3352102;
   W_i[14,27] := 0.03507431;
   W_i[14,28] := -0.1267896;
   W_i[14,29] := 0.1670964;
   W_i[14,30] := -0.0505274;
   W_i[14,31] := -0.1180039;
   W_i[14,32] := -0.0957516;
   W_i[14,33] := -0.01452094;
   W_i[14,34] := 0.00625472;
   W_i[14,35] := -0.1287756;
   W_i[14,36] := -0.06069501;
   W_i[14,37] := -0.2287704;
   W_i[14,38] := 0.1723173;
   W_i[14,39] := 1.048311;
   W_i[15,0] := 0.04376059;
   W_i[15,1] := -0.02296846;
   W_i[15,2] := 0.01713722;
   W_i[15,3] := 0.1710745;
   W_i[15,4] := 0.1736928;
   W_i[15,5] := -0.01825109;
   W_i[15,6] := -0.02258963;
   W_i[15,7] := 0.02190229;
   W_i[15,8] := -0.03702974;
   W_i[15,9] := -0.03196403;
   W_i[15,10] := 0.0826442;
   W_i[15,11] := 0.05920084;
   W_i[15,12] := -0.4280593;
   W_i[15,13] := -0.1717298;
   W_i[15,14] := 0.02115602;
   W_i[15,15] := -0.00198027;
   W_i[15,16] := 0.02912534;
   W_i[15,17] := -0.07075519;
   W_i[15,18] := -0.1174446;
   W_i[15,19] := 0.3068856;
   W_i[15,20] := 0.04301663;
   W_i[15,21] := 0.2163539;
   W_i[15,22] := -0.08966552;
   W_i[15,23] := 0.07217173;
   W_i[15,24] := -0.5324492;
   W_i[15,25] := -0.1716945;
   W_i[15,26] := -0.00556448;
   W_i[15,27] := -0.1629407;
   W_i[15,28] := 0.0326442;
   W_i[15,29] := 0.01573053;
   W_i[15,30] := -0.03329111;
   W_i[15,31] := -0.01247096;
   W_i[15,32] := 0.2100068;
   W_i[15,33] := 0.1504364;
   W_i[15,34] := -0.1697979;
   W_i[15,35] := 0.00504174;
   W_i[15,36] := 0.00267995;
   W_i[15,37] := -0.06215737;
   W_i[15,38] := 0.2148149;
   W_i[15,39] := 0.07231134;
   W_f[0,0] := -0.02091779;
   W_f[0,1] := -0.01810063;
   W_f[0,2] := 0.210087;
   W_f[0,3] := 0.09207959;
   W_f[0,4] := -0.106951;
   W_f[0,5] := -0.03611851;
   W_f[0,6] := 0.03397696;
   W_f[0,7] := 0.1654486;
   W_f[0,8] := -0.05997881;
   W_f[0,9] := -0.00453302;
   W_f[0,10] := 0.03307042;
   W_f[0,11] := 0.1420249;
   W_f[0,12] := 0.08012222;
   W_f[0,13] := -0.01528266;
   W_f[0,14] := -0.1520115;
   W_f[0,15] := -0.1571838;
   W_f[0,16] := -0.08413183;
   W_f[0,17] := 0.202225;
   W_f[0,18] := -0.01353853;
   W_f[0,19] := 0.02782044;
   W_f[0,20] := -0.04748038;
   W_f[0,21] := 0.1830429;
   W_f[0,22] := 0.312574;
   W_f[0,23] := -0.06208337;
   W_f[0,24] := 1.601337;
   W_f[0,25] := 1.519568;
   W_f[0,26] := 0.00266673;
   W_f[0,27] := 0.1218089;
   W_f[0,28] := 0.04435247;
   W_f[0,29] := 0.03200248;
   W_f[0,30] := 0.3833835;
   W_f[0,31] := 0.04435838;
   W_f[0,32] := 0.3068092;
   W_f[0,33] := 0.1323125;
   W_f[0,34] := 1.357195;
   W_f[0,35] := 0.3687007;
   W_f[0,36] := 0.08067872;
   W_f[0,37] := 0.2129946;
   W_f[0,38] := -0.02734181;
   W_f[0,39] := 0.07611577;
   W_f[1,0] := -0.388171;
   W_f[1,1] := 0.0277961;
   W_f[1,2] := -0.2651086;
   W_f[1,3] := -0.07072625;
   W_f[1,4] := 0.1196625;
   W_f[1,5] := 0.1200041;
   W_f[1,6] := -0.5084692;
   W_f[1,7] := -0.1336109;
   W_f[1,8] := -0.1377796;
   W_f[1,9] := -0.08736181;
   W_f[1,10] := 0.3113477;
   W_f[1,11] := 0.08504082;
   W_f[1,12] := 0.2114833;
   W_f[1,13] := -0.1354954;
   W_f[1,14] := -0.1227995;
   W_f[1,15] := 0.05185516;
   W_f[1,16] := -0.1474537;
   W_f[1,17] := 0.05817819;
   W_f[1,18] := 1.081658;
   W_f[1,19] := 0.1838115;
   W_f[1,20] := 0.2874206;
   W_f[1,21] := -0.2731599;
   W_f[1,22] := 0.08855448;
   W_f[1,23] := -0.09573217;
   W_f[1,24] := -0.3668332;
   W_f[1,25] := -0.6991156;
   W_f[1,26] := 0.07979747;
   W_f[1,27] := -0.1754114;
   W_f[1,28] := -0.2455159;
   W_f[1,29] := 0.1498487;
   W_f[1,30] := 0.02324941;
   W_f[1,31] := 0.07932284;
   W_f[1,32] := -0.1244244;
   W_f[1,33] := 0.02366536;
   W_f[1,34] := 0.1374529;
   W_f[1,35] := 0.4630612;
   W_f[1,36] := -0.2267325;
   W_f[1,37] := 0.07258049;
   W_f[1,38] := 0.4229668;
   W_f[1,39] := 0.1492153;
   W_f[2,0] := -0.01982149;
   W_f[2,1] := 0.03324119;
   W_f[2,2] := -0.04425151;
   W_f[2,3] := 0.08356856;
   W_f[2,4] := -0.00266197;
   W_f[2,5] := -0.01017811;
   W_f[2,6] := -0.03237398;
   W_f[2,7] := -0.00609645;
   W_f[2,8] := -0.04705935;
   W_f[2,9] := 0.03853706;
   W_f[2,10] := 0.0314042;
   W_f[2,11] := -0.1204331;
   W_f[2,12] := 0.2691576;
   W_f[2,13] := 0.04188414;
   W_f[2,14] := 0.1063143;
   W_f[2,15] := 0.05646345;
   W_f[2,16] := 0.1619761;
   W_f[2,17] := 0.2140286;
   W_f[2,18] := -0.09279267;
   W_f[2,19] := -0.0057711;
   W_f[2,20] := -0.03028176;
   W_f[2,21] := -0.05153098;
   W_f[2,22] := -0.1101711;
   W_f[2,23] := -0.01419843;
   W_f[2,24] := -0.6308476;
   W_f[2,25] := -0.4115897;
   W_f[2,26] := -0.1494104;
   W_f[2,27] := 0.04505387;
   W_f[2,28] := 0.09163468;
   W_f[2,29] := 0.2042337;
   W_f[2,30] := -0.05021087;
   W_f[2,31] := -0.05815214;
   W_f[2,32] := -0.04207016;
   W_f[2,33] := 0.2173674;
   W_f[2,34] := 0.6430734;
   W_f[2,35] := -0.1955237;
   W_f[2,36] := -0.05630085;
   W_f[2,37] := 0.0053133;
   W_f[2,38] := -0.1228282;
   W_f[2,39] := 0.5455168;
   W_f[3,0] := -0.00758014;
   W_f[3,1] := 0.00559481;
   W_f[3,2] := 0.04034248;
   W_f[3,3] := 0.02266315;
   W_f[3,4] := -0.09543922;
   W_f[3,5] := 0.03211372;
   W_f[3,6] := 0.07329436;
   W_f[3,7] := -0.04057672;
   W_f[3,8] := -0.09598581;
   W_f[3,9] := -0.00159119;
   W_f[3,10] := 0.00039486;
   W_f[3,11] := -0.00788106;
   W_f[3,12] := -0.06210583;
   W_f[3,13] := -0.01413072;
   W_f[3,14] := -0.2401386;
   W_f[3,15] := -0.07759018;
   W_f[3,16] := 0.0436046;
   W_f[3,17] := -0.2098783;
   W_f[3,18] := 0.1486036;
   W_f[3,19] := -0.02982033;
   W_f[3,20] := -0.08417022;
   W_f[3,21] := 0.08484244;
   W_f[3,22] := 0.3341856;
   W_f[3,23] := -0.01567571;
   W_f[3,24] := 1.093444;
   W_f[3,25] := 0.9772373;
   W_f[3,26] := -0.1362202;
   W_f[3,27] := -0.0995613;
   W_f[3,28] := 0.00698416;
   W_f[3,29] := 0.0005413;
   W_f[3,30] := 0.2605347;
   W_f[3,31] := -0.09947061;
   W_f[3,32] := 0.2628707;
   W_f[3,33] := 0.00611334;
   W_f[3,34] := 1.38905;
   W_f[3,35] := -0.1434975;
   W_f[3,36] := -0.00342261;
   W_f[3,37] := -0.06542191;
   W_f[3,38] := 0.1048234;
   W_f[3,39] := 0.1138595;
   W_f[4,0] := 0.2867894;
   W_f[4,1] := -0.1455002;
   W_f[4,2] := 0.2030114;
   W_f[4,3] := -0.1528496;
   W_f[4,4] := -0.1193404;
   W_f[4,5] := -0.06261637;
   W_f[4,6] := -0.09047025;
   W_f[4,7] := -0.02217131;
   W_f[4,8] := 0.3289314;
   W_f[4,9] := -0.5019218;
   W_f[4,10] := -0.02496753;
   W_f[4,11] := -0.02753776;
   W_f[4,12] := -0.3154772;
   W_f[4,13] := -0.04408565;
   W_f[4,14] := 0.05384916;
   W_f[4,15] := -0.3253689;
   W_f[4,16] := -0.01380023;
   W_f[4,17] := -0.121247;
   W_f[4,18] := 0.6214666;
   W_f[4,19] := 0.01393374;
   W_f[4,20] := 0.04359875;
   W_f[4,21] := 0.1630262;
   W_f[4,22] := -0.2102474;
   W_f[4,23] := -0.1291176;
   W_f[4,24] := -0.0868592;
   W_f[4,25] := -0.03674764;
   W_f[4,26] := 0.3087266;
   W_f[4,27] := 0.03806484;
   W_f[4,28] := 0.01020021;
   W_f[4,29] := -0.1519751;
   W_f[4,30] := 0.05839425;
   W_f[4,31] := -0.01564794;
   W_f[4,32] := -0.1834329;
   W_f[4,33] := 0.02443381;
   W_f[4,34] := 0.2140227;
   W_f[4,35] := 0.1936068;
   W_f[4,36] := 0.09160208;
   W_f[4,37] := 0.06046678;
   W_f[4,38] := -0.08968955;
   W_f[4,39] := -0.03439303;
   W_f[5,0] := -0.3995713;
   W_f[5,1] := -0.4650751;
   W_f[5,2] := -0.2646359;
   W_f[5,3] := -0.08991144;
   W_f[5,4] := -0.1660275;
   W_f[5,5] := 0.3650228;
   W_f[5,6] := -0.03514609;
   W_f[5,7] := -0.0638742;
   W_f[5,8] := 0.1263784;
   W_f[5,9] := 0.1945071;
   W_f[5,10] := -0.07852599;
   W_f[5,11] := -0.2437045;
   W_f[5,12] := -0.06879438;
   W_f[5,13] := 0.2681186;
   W_f[5,14] := 0.01808503;
   W_f[5,15] := -0.1007093;
   W_f[5,16] := 0.3104329;
   W_f[5,17] := -0.03764273;
   W_f[5,18] := -0.05466426;
   W_f[5,19] := -0.1028605;
   W_f[5,20] := -0.1891315;
   W_f[5,21] := -0.062895;
   W_f[5,22] := 0.2626143;
   W_f[5,23] := 0.1165986;
   W_f[5,24] := 2.139313;
   W_f[5,25] := 2.362694;
   W_f[5,26] := -0.4129075;
   W_f[5,27] := 0.08711372;
   W_f[5,28] := -0.06960621;
   W_f[5,29] := -0.1088286;
   W_f[5,30] := 0.02405319;
   W_f[5,31] := -0.02791615;
   W_f[5,32] := -0.03174478;
   W_f[5,33] := -0.2259803;
   W_f[5,34] := 0.02213258;
   W_f[5,35] := 0.06206211;
   W_f[5,36] := -0.220625;
   W_f[5,37] := 0.2029873;
   W_f[5,38] := 0.03730853;
   W_f[5,39] := -0.1644827;
   W_f[6,0] := 0.09157378;
   W_f[6,1] := -0.106003;
   W_f[6,2] := 0.01516851;
   W_f[6,3] := -0.09814398;
   W_f[6,4] := -0.02060772;
   W_f[6,5] := -0.1166353;
   W_f[6,6] := 0.1760547;
   W_f[6,7] := 0.1404383;
   W_f[6,8] := -0.06626645;
   W_f[6,9] := 0.0325418;
   W_f[6,10] := -0.03667779;
   W_f[6,11] := 0.03295979;
   W_f[6,12] := 0.1345612;
   W_f[6,13] := 0.1752782;
   W_f[6,14] := 0.06438499;
   W_f[6,15] := -0.1272106;
   W_f[6,16] := -0.2878087;
   W_f[6,17] := 0.1161476;
   W_f[6,18] := -0.2311435;
   W_f[6,19] := -0.07521003;
   W_f[6,20] := -0.1416016;
   W_f[6,21] := 0.1268703;
   W_f[6,22] := 0.3855781;
   W_f[6,23] := -0.1290094;
   W_f[6,24] := 1.145507;
   W_f[6,25] := 1.206513;
   W_f[6,26] := 0.01718643;
   W_f[6,27] := -0.2014013;
   W_f[6,28] := -0.03907681;
   W_f[6,29] := -1.031836;
   W_f[6,30] := 0.1329869;
   W_f[6,31] := -0.05304611;
   W_f[6,32] := 0.2754238;
   W_f[6,33] := 0.484001;
   W_f[6,34] := 0.8730348;
   W_f[6,35] := -0.2791631;
   W_f[6,36] := 0.09285419;
   W_f[6,37] := -0.00086587;
   W_f[6,38] := 0.2140355;
   W_f[6,39] := 0.01036415;
   W_f[7,0] := -0.00185265;
   W_f[7,1] := 0.07858364;
   W_f[7,2] := 0.00610039;
   W_f[7,3] := 0.06575946;
   W_f[7,4] := -0.0810083;
   W_f[7,5] := 0.00321988;
   W_f[7,6] := 0.07597861;
   W_f[7,7] := -0.1263862;
   W_f[7,8] := 0.1467239;
   W_f[7,9] := 0.04145058;
   W_f[7,10] := 0.03552409;
   W_f[7,11] := -0.4200411;
   W_f[7,12] := 0.2535799;
   W_f[7,13] := -0.08330481;
   W_f[7,14] := -0.08974353;
   W_f[7,15] := -0.1051762;
   W_f[7,16] := -0.3822444;
   W_f[7,17] := -0.4579986;
   W_f[7,18] := -0.06309059;
   W_f[7,19] := -0.3079986;
   W_f[7,20] := -0.08522949;
   W_f[7,21] := -0.06581733;
   W_f[7,22] := 0.2580513;
   W_f[7,23] := 0.02311642;
   W_f[7,24] := 0.9095069;
   W_f[7,25] := 1.188896;
   W_f[7,26] := -0.1154661;
   W_f[7,27] := -0.1087225;
   W_f[7,28] := -0.08876549;
   W_f[7,29] := 0.00109644;
   W_f[7,30] := 0.2337219;
   W_f[7,31] := -0.1376933;
   W_f[7,32] := 0.1659716;
   W_f[7,33] := 0.04170239;
   W_f[7,34] := 1.311337;
   W_f[7,35] := -0.1188877;
   W_f[7,36] := 0.04907094;
   W_f[7,37] := 0.1402612;
   W_f[7,38] := 0.1255982;
   W_f[7,39] := -1.274189;
   W_f[8,0] := 0.12556;
   W_f[8,1] := -0.1031576;
   W_f[8,2] := 0.03551091;
   W_f[8,3] := -0.03898631;
   W_f[8,4] := -0.1320676;
   W_f[8,5] := 0.07454634;
   W_f[8,6] := 0.1020655;
   W_f[8,7] := 0.01262685;
   W_f[8,8] := -0.00534601;
   W_f[8,9] := -0.00536494;
   W_f[8,10] := -0.04092396;
   W_f[8,11] := -0.3869237;
   W_f[8,12] := 0.03422466;
   W_f[8,13] := 0.02580789;
   W_f[8,14] := 0.2689887;
   W_f[8,15] := -0.2494489;
   W_f[8,16] := -0.02722716;
   W_f[8,17] := -0.1010804;
   W_f[8,18] := 0.5424435;
   W_f[8,19] := -0.2312066;
   W_f[8,20] := -0.04103015;
   W_f[8,21] := -0.1674081;
   W_f[8,22] := 0.1389381;
   W_f[8,23] := -0.04656294;
   W_f[8,24] := 0.531742;
   W_f[8,25] := 0.7430941;
   W_f[8,26] := -0.00084738;
   W_f[8,27] := -0.04600925;
   W_f[8,28] := -0.1588;
   W_f[8,29] := 0.08535929;
   W_f[8,30] := 0.1022129;
   W_f[8,31] := -0.03335671;
   W_f[8,32] := 0.03138823;
   W_f[8,33] := -0.02403146;
   W_f[8,34] := 0.8330596;
   W_f[8,35] := -0.07033388;
   W_f[8,36] := -0.1749986;
   W_f[8,37] := 0.0922937;
   W_f[8,38] := -0.1766868;
   W_f[8,39] := 0.141985;
   W_f[9,0] := -0.08198071;
   W_f[9,1] := 0.03835172;
   W_f[9,2] := 1.020265;
   W_f[9,3] := -0.1529395;
   W_f[9,4] := -0.1617989;
   W_f[9,5] := 0.03072036;
   W_f[9,6] := -0.09759208;
   W_f[9,7] := -0.07946933;
   W_f[9,8] := -0.6549187;
   W_f[9,9] := 0.2455487;
   W_f[9,10] := -0.00084776;
   W_f[9,11] := -0.02393647;
   W_f[9,12] := -0.1103576;
   W_f[9,13] := 0.05757844;
   W_f[9,14] := 0.00252463;
   W_f[9,15] := -0.04278835;
   W_f[9,16] := -0.01363701;
   W_f[9,17] := 0.03181182;
   W_f[9,18] := 0.2954217;
   W_f[9,19] := 0.1868071;
   W_f[9,20] := -0.1459624;
   W_f[9,21] := 0.04626612;
   W_f[9,22] := -0.4959656;
   W_f[9,23] := -0.298828;
   W_f[9,24] := -0.05025842;
   W_f[9,25] := -0.2492222;
   W_f[9,26] := 0.2277043;
   W_f[9,27] := -0.077122;
   W_f[9,28] := -0.1601862;
   W_f[9,29] := -0.360285;
   W_f[9,30] := -0.1589459;
   W_f[9,31] := 0.07634185;
   W_f[9,32] := -0.1424809;
   W_f[9,33] := 0.4724371;
   W_f[9,34] := 0.3722708;
   W_f[9,35] := 0.08862774;
   W_f[9,36] := 0.1802045;
   W_f[9,37] := -0.4637271;
   W_f[9,38] := 0.1014335;
   W_f[9,39] := 0.0325746;
   W_f[10,0] := 0.01476683;
   W_f[10,1] := 0.0891594;
   W_f[10,2] := 0.09493639;
   W_f[10,3] := 0.0092164;
   W_f[10,4] := -0.4010172;
   W_f[10,5] := -0.09464957;
   W_f[10,6] := -0.04691195;
   W_f[10,7] := -0.02866868;
   W_f[10,8] := -0.04315028;
   W_f[10,9] := -0.1709383;
   W_f[10,10] := -0.00073274;
   W_f[10,11] := -0.2750555;
   W_f[10,12] := 0.3360567;
   W_f[10,13] := -0.2203442;
   W_f[10,14] := 0.2416514;
   W_f[10,15] := -0.2352184;
   W_f[10,16] := -0.00154005;
   W_f[10,17] := -0.00158511;
   W_f[10,18] := 0.1191233;
   W_f[10,19] := -0.02448388;
   W_f[10,20] := -0.2385904;
   W_f[10,21] := -0.05945824;
   W_f[10,22] := 0.01714438;
   W_f[10,23] := -0.1828551;
   W_f[10,24] := 1.57859;
   W_f[10,25] := 1.894226;
   W_f[10,26] := 0.09559432;
   W_f[10,27] := -0.273827;
   W_f[10,28] := -0.2814649;
   W_f[10,29] := 0.04344108;
   W_f[10,30] := 0.08430442;
   W_f[10,31] := 0.1357144;
   W_f[10,32] := 0.03089454;
   W_f[10,33] := 0.1987186;
   W_f[10,34] := 0.1212473;
   W_f[10,35] := 0.1387797;
   W_f[10,36] := 0.2638152;
   W_f[10,37] := 0.00209056;
   W_f[10,38] := -0.08942132;
   W_f[10,39] := -0.4494387;
   W_f[11,0] := 0.04211291;
   W_f[11,1] := -0.02505053;
   W_f[11,2] := 0.08745301;
   W_f[11,3] := -0.04265523;
   W_f[11,4] := -0.2127612;
   W_f[11,5] := 0.01322894;
   W_f[11,6] := 0.1062051;
   W_f[11,7] := 0.01512342;
   W_f[11,8] := -0.07057641;
   W_f[11,9] := 0.1239847;
   W_f[11,10] := -0.1409187;
   W_f[11,11] := -0.0726796;
   W_f[11,12] := 0.00417219;
   W_f[11,13] := -0.01783882;
   W_f[11,14] := 0.01799064;
   W_f[11,15] := -0.05493079;
   W_f[11,16] := -0.05114271;
   W_f[11,17] := -0.03128599;
   W_f[11,18] := 0.03801877;
   W_f[11,19] := -0.01814952;
   W_f[11,20] := -0.09758195;
   W_f[11,21] := -0.04573784;
   W_f[11,22] := -0.03167154;
   W_f[11,23] := -0.08901857;
   W_f[11,24] := -0.2217392;
   W_f[11,25] := 0.3994405;
   W_f[11,26] := 0.0512911;
   W_f[11,27] := 0.05733421;
   W_f[11,28] := -0.1220476;
   W_f[11,29] := 0.2530152;
   W_f[11,30] := -0.01943143;
   W_f[11,31] := 0.06523979;
   W_f[11,32] := -0.1965705;
   W_f[11,33] := 0.010429;
   W_f[11,34] := 0.1933591;
   W_f[11,35] := -0.02032585;
   W_f[11,36] := -0.05446678;
   W_f[11,37] := 0.1093058;
   W_f[11,38] := -0.05791799;
   W_f[11,39] := 0.3272165;
   W_f[12,0] := 0.0583974;
   W_f[12,1] := 0.06337267;
   W_f[12,2] := 0.05269343;
   W_f[12,3] := -0.02425898;
   W_f[12,4] := 0.0733385;
   W_f[12,5] := 0.01520942;
   W_f[12,6] := 0.03044897;
   W_f[12,7] := 0.1151135;
   W_f[12,8] := 0.03681342;
   W_f[12,9] := -0.0168035;
   W_f[12,10] := 0.04408923;
   W_f[12,11] := 0.08383411;
   W_f[12,12] := -0.01220268;
   W_f[12,13] := 0.0539641;
   W_f[12,14] := -0.07032214;
   W_f[12,15] := -0.00997462;
   W_f[12,16] := -0.06021495;
   W_f[12,17] := -0.01422043;
   W_f[12,18] := -0.00584967;
   W_f[12,19] := 0.05498984;
   W_f[12,20] := -0.0921667;
   W_f[12,21] := 0.1078821;
   W_f[12,22] := 0.09067565;
   W_f[12,23] := -0.09486815;
   W_f[12,24] := -0.8760142;
   W_f[12,25] := 0.543728;
   W_f[12,26] := 0.0473772;
   W_f[12,27] := -0.1004083;
   W_f[12,28] := 0.07258554;
   W_f[12,29] := 0.07306878;
   W_f[12,30] := -0.1469819;
   W_f[12,31] := 0.01059632;
   W_f[12,32] := 0.01764544;
   W_f[12,33] := -0.04630747;
   W_f[12,34] := 0.04829778;
   W_f[12,35] := -0.00637231;
   W_f[12,36] := 0.3430251;
   W_f[12,37] := 0.1221798;
   W_f[12,38] := 0.04078831;
   W_f[12,39] := 0.02011232;
   W_f[13,0] := 0.1598776;
   W_f[13,1] := 0.08477814;
   W_f[13,2] := -0.1199006;
   W_f[13,3] := -0.2151837;
   W_f[13,4] := 0.04422749;
   W_f[13,5] := 0.1643971;
   W_f[13,6] := -0.01991516;
   W_f[13,7] := 0.01602156;
   W_f[13,8] := -0.134406;
   W_f[13,9] := 0.0432152;
   W_f[13,10] := 0.1258369;
   W_f[13,11] := 0.03486055;
   W_f[13,12] := 0.1840334;
   W_f[13,13] := 0.05531228;
   W_f[13,14] := -0.05205994;
   W_f[13,15] := -0.1417992;
   W_f[13,16] := 0.2145569;
   W_f[13,17] := -0.03670088;
   W_f[13,18] := 0.05554622;
   W_f[13,19] := -0.0701214;
   W_f[13,20] := 0.05645064;
   W_f[13,21] := 0.04904451;
   W_f[13,22] := 0.1227407;
   W_f[13,23] := -0.1391225;
   W_f[13,24] := 1.281417;
   W_f[13,25] := 1.152952;
   W_f[13,26] := 0.02036783;
   W_f[13,27] := 6.46E-06;
   W_f[13,28] := 0.05594068;
   W_f[13,29] := 0.1138421;
   W_f[13,30] := 0.2391586;
   W_f[13,31] := 0.04423625;
   W_f[13,32] := 0.3790507;
   W_f[13,33] := 0.01350218;
   W_f[13,34] := 0.907777;
   W_f[13,35] := -0.01705103;
   W_f[13,36] := 0.08728553;
   W_f[13,37] := 0.1376872;
   W_f[13,38] := 0.05409899;
   W_f[13,39] := 0.5876323;
   W_f[14,0] := -0.1830878;
   W_f[14,1] := 0.00258858;
   W_f[14,2] := -0.05409549;
   W_f[14,3] := 0.4265317;
   W_f[14,4] := -0.1661472;
   W_f[14,5] := -0.06032855;
   W_f[14,6] := 0.09126755;
   W_f[14,7] := -0.1622344;
   W_f[14,8] := -0.0415544;
   W_f[14,9] := -0.03031821;
   W_f[14,10] := -0.07388397;
   W_f[14,11] := -0.1665972;
   W_f[14,12] := 0.1223991;
   W_f[14,13] := -0.1334893;
   W_f[14,14] := -0.06961614;
   W_f[14,15] := -0.04957403;
   W_f[14,16] := 0.0298849;
   W_f[14,17] := -0.1339389;
   W_f[14,18] := -0.04285705;
   W_f[14,19] := -0.08629614;
   W_f[14,20] := -0.1532967;
   W_f[14,21] := 0.04812383;
   W_f[14,22] := -0.03088393;
   W_f[14,23] := -0.04624541;
   W_f[14,24] := -0.07781153;
   W_f[14,25] := -0.8319644;
   W_f[14,26] := 0.1015401;
   W_f[14,27] := 0.04807844;
   W_f[14,28] := 0.08697836;
   W_f[14,29] := -0.3099394;
   W_f[14,30] := 0.02526759;
   W_f[14,31] := 0.06875665;
   W_f[14,32] := 0.05270454;
   W_f[14,33] := 0.08052166;
   W_f[14,34] := 0.07316659;
   W_f[14,35] := -0.2259305;
   W_f[14,36] := -0.0360414;
   W_f[14,37] := -0.1107528;
   W_f[14,38] := 0.1422287;
   W_f[14,39] := 0.1191253;
   W_f[15,0] := 0.06860624;
   W_f[15,1] := 0.2116713;
   W_f[15,2] := -0.1070077;
   W_f[15,3] := -0.1796377;
   W_f[15,4] := 0.06190439;
   W_f[15,5] := 0.1118638;
   W_f[15,6] := 0.2123804;
   W_f[15,7] := 0.04805397;
   W_f[15,8] := 0.02383129;
   W_f[15,9] := -0.08112741;
   W_f[15,10] := -0.00035556;
   W_f[15,11] := -0.00759834;
   W_f[15,12] := 0.04278949;
   W_f[15,13] := -0.01575772;
   W_f[15,14] := -0.06780741;
   W_f[15,15] := 0.07988951;
   W_f[15,16] := 0.3583542;
   W_f[15,17] := -0.1143483;
   W_f[15,18] := 0.06204842;
   W_f[15,19] := -0.1630864;
   W_f[15,20] := -0.08014372;
   W_f[15,21] := 0.09970582;
   W_f[15,22] := -0.01455338;
   W_f[15,23] := -0.09048357;
   W_f[15,24] := 1.480857;
   W_f[15,25] := 1.437098;
   W_f[15,26] := -0.04126001;
   W_f[15,27] := 0.03295555;
   W_f[15,28] := -0.0889762;
   W_f[15,29] := 0.1496947;
   W_f[15,30] := 0.1286354;
   W_f[15,31] := -0.01891266;
   W_f[15,32] := -0.08377147;
   W_f[15,33] := 0.04984247;
   W_f[15,34] := 0.7321002;
   W_f[15,35] := -0.07470711;
   W_f[15,36] := 0.01260767;
   W_f[15,37] := -0.02138078;
   W_f[15,38] := 0.01280809;
   W_f[15,39] := 0.1211099;
   W_g[0,0] := 0.1320454;
   W_g[0,1] := -0.07179091;
   W_g[0,2] := 0.1304129;
   W_g[0,3] := -0.01710966;
   W_g[0,4] := 0.08717188;
   W_g[0,5] := -0.03005558;
   W_g[0,6] := 0.02608494;
   W_g[0,7] := -0.02178418;
   W_g[0,8] := -0.02002059;
   W_g[0,9] := -0.01907159;
   W_g[0,10] := -0.07584066;
   W_g[0,11] := -0.0276128;
   W_g[0,12] := -0.03857584;
   W_g[0,13] := -0.01737243;
   W_g[0,14] := -0.1033841;
   W_g[0,15] := -0.00566125;
   W_g[0,16] := -0.01846444;
   W_g[0,17] := -0.09568264;
   W_g[0,18] := 0.01344434;
   W_g[0,19] := -0.04545733;
   W_g[0,20] := -0.07012872;
   W_g[0,21] := -0.2265758;
   W_g[0,22] := -0.0013438;
   W_g[0,23] := 0.0140279;
   W_g[0,24] := 0.05787951;
   W_g[0,25] := 0.3332284;
   W_g[0,26] := 0.1338745;
   W_g[0,27] := -0.284954;
   W_g[0,28] := 0.08640742;
   W_g[0,29] := 0.00553245;
   W_g[0,30] := 0.00379307;
   W_g[0,31] := 0.00939364;
   W_g[0,32] := -0.0225928;
   W_g[0,33] := -0.03415785;
   W_g[0,34] := 0.4156659;
   W_g[0,35] := -0.02096383;
   W_g[0,36] := -0.0417503;
   W_g[0,37] := -0.04161927;
   W_g[0,38] := 0.04176929;
   W_g[0,39] := -0.02666814;
   W_g[1,0] := 0.1003403;
   W_g[1,1] := 0.02818905;
   W_g[1,2] := 0.08966444;
   W_g[1,3] := 0.02384869;
   W_g[1,4] := -0.00957148;
   W_g[1,5] := 0.0225874;
   W_g[1,6] := 0.2189841;
   W_g[1,7] := 0.03297459;
   W_g[1,8] := 0.02741309;
   W_g[1,9] := 0.03524271;
   W_g[1,10] := -0.09459055;
   W_g[1,11] := 0.00226336;
   W_g[1,12] := -0.03214818;
   W_g[1,13] := 0.09925831;
   W_g[1,14] := 0.03271784;
   W_g[1,15] := -0.00993501;
   W_g[1,16] := 0.04625125;
   W_g[1,17] := -0.01382133;
   W_g[1,18] := 0.141697;
   W_g[1,19] := -0.06103647;
   W_g[1,20] := -0.2125344;
   W_g[1,21] := 0.1183949;
   W_g[1,22] := -0.01691977;
   W_g[1,23] := 0.05358729;
   W_g[1,24] := -0.3285331;
   W_g[1,25] := -0.4942485;
   W_g[1,26] := -0.08112237;
   W_g[1,27] := 0.1249737;
   W_g[1,28] := 0.1749274;
   W_g[1,29] := 0.05923015;
   W_g[1,30] := -0.03070631;
   W_g[1,31] := -0.0160953;
   W_g[1,32] := 0.0128262;
   W_g[1,33] := 0.00597268;
   W_g[1,34] := -0.4454135;
   W_g[1,35] := 0.04373179;
   W_g[1,36] := 0.07117015;
   W_g[1,37] := -0.05477969;
   W_g[1,38] := -0.1148913;
   W_g[1,39] := -0.05603904;
   W_g[2,0] := -0.03656583;
   W_g[2,1] := 0.08601304;
   W_g[2,2] := -0.02144271;
   W_g[2,3] := -0.00415884;
   W_g[2,4] := 0.05374509;
   W_g[2,5] := 0.01513857;
   W_g[2,6] := 0.00031003;
   W_g[2,7] := -0.00429267;
   W_g[2,8] := 0.0024794;
   W_g[2,9] := -0.02802207;
   W_g[2,10] := 0.00567887;
   W_g[2,11] := 0.07285577;
   W_g[2,12] := 0.06949551;
   W_g[2,13] := -0.06609099;
   W_g[2,14] := 0.02675425;
   W_g[2,15] := 0.05979875;
   W_g[2,16] := 0.1882337;
   W_g[2,17] := 0.1013563;
   W_g[2,18] := -0.01730143;
   W_g[2,19] := 0.07176489;
   W_g[2,20] := -0.00487325;
   W_g[2,21] := -0.01244247;
   W_g[2,22] := 0.07138075;
   W_g[2,23] := -0.08855219;
   W_g[2,24] := 0.6691746;
   W_g[2,25] := 0.4066471;
   W_g[2,26] := 0.05317146;
   W_g[2,27] := -0.03753066;
   W_g[2,28] := 0.04217075;
   W_g[2,29] := -0.08696262;
   W_g[2,30] := 0.0727913;
   W_g[2,31] := 0.04612178;
   W_g[2,32] := 0.06409022;
   W_g[2,33] := 0.01605693;
   W_g[2,34] := 0.1564854;
   W_g[2,35] := 0.1177737;
   W_g[2,36] := -0.03577918;
   W_g[2,37] := -0.02626175;
   W_g[2,38] := -0.2925088;
   W_g[2,39] := -0.1730511;
   W_g[3,0] := 0.0353583;
   W_g[3,1] := -0.1049412;
   W_g[3,2] := 0.03618518;
   W_g[3,3] := -0.03134191;
   W_g[3,4] := -0.2461421;
   W_g[3,5] := 0.1266218;
   W_g[3,6] := 0.06337537;
   W_g[3,7] := -0.035273;
   W_g[3,8] := -0.03651504;
   W_g[3,9] := -0.03074392;
   W_g[3,10] := -0.05727396;
   W_g[3,11] := -0.02935094;
   W_g[3,12] := -0.03621458;
   W_g[3,13] := -0.01833671;
   W_g[3,14] := -0.1685012;
   W_g[3,15] := -0.00882464;
   W_g[3,16] := -0.02389451;
   W_g[3,17] := -0.07828564;
   W_g[3,18] := 0.02588245;
   W_g[3,19] := -0.04996347;
   W_g[3,20] := -0.03450434;
   W_g[3,21] := 0.08713186;
   W_g[3,22] := 0.04250673;
   W_g[3,23] := 0.0231547;
   W_g[3,24] := 0.2406025;
   W_g[3,25] := -0.04010823;
   W_g[3,26] := -0.04215078;
   W_g[3,27] := 0.0426458;
   W_g[3,28] := -0.2496434;
   W_g[3,29] := -0.019585;
   W_g[3,30] := 0.03981116;
   W_g[3,31] := 0.05331163;
   W_g[3,32] := 0.02955173;
   W_g[3,33] := 0.03688915;
   W_g[3,34] := -0.07779746;
   W_g[3,35] := 0.04131736;
   W_g[3,36] := -0.09415401;
   W_g[3,37] := 0.02781735;
   W_g[3,38] := -0.01530841;
   W_g[3,39] := -0.103936;
   W_g[4,0] := 0.07740436;
   W_g[4,1] := -0.07530216;
   W_g[4,2] := 0.08100316;
   W_g[4,3] := -0.03866265;
   W_g[4,4] := -0.124116;
   W_g[4,5] := -0.06374057;
   W_g[4,6] := -0.06540763;
   W_g[4,7] := -0.05087971;
   W_g[4,8] := -0.02486523;
   W_g[4,9] := -0.00432705;
   W_g[4,10] := -0.02001161;
   W_g[4,11] := -0.2260205;
   W_g[4,12] := -0.2710404;
   W_g[4,13] := -0.04622217;
   W_g[4,14] := 0.03693646;
   W_g[4,15] := -0.2228938;
   W_g[4,16] := -0.03339233;
   W_g[4,17] := -0.1039548;
   W_g[4,18] := -0.6776975;
   W_g[4,19] := -0.1070111;
   W_g[4,20] := -0.00507321;
   W_g[4,21] := 0.06153874;
   W_g[4,22] := -0.05829039;
   W_g[4,23] := -0.03399877;
   W_g[4,24] := 0.02580869;
   W_g[4,25] := -0.05605169;
   W_g[4,26] := 0.02870816;
   W_g[4,27] := 0.09912029;
   W_g[4,28] := -0.08475526;
   W_g[4,29] := 0.02515182;
   W_g[4,30] := -0.06613169;
   W_g[4,31] := -0.01619294;
   W_g[4,32] := -0.07978069;
   W_g[4,33] := -0.02161121;
   W_g[4,34] := -0.01309834;
   W_g[4,35] := -0.0583593;
   W_g[4,36] := 0.02740471;
   W_g[4,37] := -0.06427267;
   W_g[4,38] := -0.1435904;
   W_g[4,39] := -0.04779189;
   W_g[5,0] := 0.07845761;
   W_g[5,1] := 0.122912;
   W_g[5,2] := 0.09020026;
   W_g[5,3] := -0.05951332;
   W_g[5,4] := -0.1863579;
   W_g[5,5] := -0.6706011;
   W_g[5,6] := -0.09371807;
   W_g[5,7] := -0.0624865;
   W_g[5,8] := -0.05328716;
   W_g[5,9] := -0.05699488;
   W_g[5,10] := -0.2100334;
   W_g[5,11] := -0.04094445;
   W_g[5,12] := -0.03951516;
   W_g[5,13] := 0.01896183;
   W_g[5,14] := 0.05772699;
   W_g[5,15] := -0.03484442;
   W_g[5,16] := -0.08915464;
   W_g[5,17] := -0.03359089;
   W_g[5,18] := 0.05330428;
   W_g[5,19] := -0.04913564;
   W_g[5,20] := -0.02437795;
   W_g[5,21] := -0.03660732;
   W_g[5,22] := 0.05388405;
   W_g[5,23] := 0.03580718;
   W_g[5,24] := 0.6679524;
   W_g[5,25] := 0.3846368;
   W_g[5,26] := 0.03221167;
   W_g[5,27] := -0.09449711;
   W_g[5,28] := -0.2133287;
   W_g[5,29] := -0.1070377;
   W_g[5,30] := 0.0486634;
   W_g[5,31] := 0.04555348;
   W_g[5,32] := 0.03119684;
   W_g[5,33] := 0.02472051;
   W_g[5,34] := -0.00109696;
   W_g[5,35] := 0.00976827;
   W_g[5,36] := -0.04086661;
   W_g[5,37] := 0.01402589;
   W_g[5,38] := 0.01088466;
   W_g[5,39] := 0.05395384;
   W_g[6,0] := -0.09459254;
   W_g[6,1] := -0.3465888;
   W_g[6,2] := -0.1204124;
   W_g[6,3] := 0.1131463;
   W_g[6,4] := 0.07203985;
   W_g[6,5] := -0.09553758;
   W_g[6,6] := -0.03457065;
   W_g[6,7] := 0.1258941;
   W_g[6,8] := 0.09656766;
   W_g[6,9] := 0.1205588;
   W_g[6,10] := 0.01646312;
   W_g[6,11] := -0.06715041;
   W_g[6,12] := -0.08268934;
   W_g[6,13] := -0.01733059;
   W_g[6,14] := 0.05910295;
   W_g[6,15] := -0.07129493;
   W_g[6,16] := -0.06239159;
   W_g[6,17] := -0.06886618;
   W_g[6,18] := 0.04810062;
   W_g[6,19] := -0.0965384;
   W_g[6,20] := 0.1695917;
   W_g[6,21] := -0.00798076;
   W_g[6,22] := 0.00821575;
   W_g[6,23] := 0.1049357;
   W_g[6,24] := 0.06085224;
   W_g[6,25] := 0.05369381;
   W_g[6,26] := -0.0201011;
   W_g[6,27] := 0.00523888;
   W_g[6,28] := -0.05049808;
   W_g[6,29] := 0.04111513;
   W_g[6,30] := 0.01227053;
   W_g[6,31] := 0.0204126;
   W_g[6,32] := -0.00532885;
   W_g[6,33] := -0.00633689;
   W_g[6,34] := -0.01163891;
   W_g[6,35] := 0.0326525;
   W_g[6,36] := -0.08721739;
   W_g[6,37] := 0.02508505;
   W_g[6,38] := -0.1394214;
   W_g[6,39] := -0.03058173;
   W_g[7,0] := 0.1329033;
   W_g[7,1] := -0.2278838;
   W_g[7,2] := 0.1442183;
   W_g[7,3] := -0.04011448;
   W_g[7,4] := -0.0098335;
   W_g[7,5] := 0.06002469;
   W_g[7,6] := 0.01148172;
   W_g[7,7] := -0.03318439;
   W_g[7,8] := -0.04474748;
   W_g[7,9] := -0.03664961;
   W_g[7,10] := -0.05171043;
   W_g[7,11] := 0.1588942;
   W_g[7,12] := 0.1881699;
   W_g[7,13] := 0.03320323;
   W_g[7,14] := 0.08849441;
   W_g[7,15] := 0.1089842;
   W_g[7,16] := -0.1042355;
   W_g[7,17] := 0.2178806;
   W_g[7,18] := -0.09352972;
   W_g[7,19] := 0.2286143;
   W_g[7,20] := 0.01804306;
   W_g[7,21] := 0.02883035;
   W_g[7,22] := 0.02334912;
   W_g[7,23] := 0.0097255;
   W_g[7,24] := 0.09000973;
   W_g[7,25] := 0.2379663;
   W_g[7,26] := -0.00529223;
   W_g[7,27] := 0.02389492;
   W_g[7,28] := 0.01771568;
   W_g[7,29] := 0.03995743;
   W_g[7,30] := 0.0237428;
   W_g[7,31] := 0.00652028;
   W_g[7,32] := 0.0237922;
   W_g[7,33] := 0.01227521;
   W_g[7,34] := -0.02105843;
   W_g[7,35] := 0.02154919;
   W_g[7,36] := -0.01575272;
   W_g[7,37] := -0.01810107;
   W_g[7,38] := -0.00772995;
   W_g[7,39] := -0.2820103;
   W_g[8,0] := 0.01713815;
   W_g[8,1] := -0.00229361;
   W_g[8,2] := 0.01726119;
   W_g[8,3] := -0.02061658;
   W_g[8,4] := -0.04641379;
   W_g[8,5] := 0.04689364;
   W_g[8,6] := 0.00514349;
   W_g[8,7] := -0.02527735;
   W_g[8,8] := -0.02019661;
   W_g[8,9] := -0.01965989;
   W_g[8,10] := -0.02106753;
   W_g[8,11] := -0.1810846;
   W_g[8,12] := -0.1747753;
   W_g[8,13] := -0.07262667;
   W_g[8,14] := 0.09604074;
   W_g[8,15] := -0.2233989;
   W_g[8,16] := -0.01457437;
   W_g[8,17] := 0.1895211;
   W_g[8,18] := 0.09061687;
   W_g[8,19] := -0.1659747;
   W_g[8,20] := -0.02462232;
   W_g[8,21] := -0.0811555;
   W_g[8,22] := 0.02058986;
   W_g[8,23] := -0.05404805;
   W_g[8,24] := -0.07197467;
   W_g[8,25] := -0.2429945;
   W_g[8,26] := 0.03455175;
   W_g[8,27] := -0.1281454;
   W_g[8,28] := -0.1244678;
   W_g[8,29] := -0.0707626;
   W_g[8,30] := 0.03440274;
   W_g[8,31] := 0.02760479;
   W_g[8,32] := -0.00320816;
   W_g[8,33] := -0.00195394;
   W_g[8,34] := -0.06706773;
   W_g[8,35] := -0.03631235;
   W_g[8,36] := -0.0461507;
   W_g[8,37] := 0.02211455;
   W_g[8,38] := 0.00710197;
   W_g[8,39] := 0.06994114;
   W_g[9,0] := -0.2685941;
   W_g[9,1] := -0.1633901;
   W_g[9,2] := -0.3089246;
   W_g[9,3] := -0.1282196;
   W_g[9,4] := 0.01028809;
   W_g[9,5] := -0.05689346;
   W_g[9,6] := 0.131765;
   W_g[9,7] := -0.1136668;
   W_g[9,8] := -0.1350522;
   W_g[9,9] := -0.1341046;
   W_g[9,10] := -0.2973659;
   W_g[9,11] := 0.03893382;
   W_g[9,12] := 0.03934914;
   W_g[9,13] := 0.01418684;
   W_g[9,14] := 0.01693503;
   W_g[9,15] := 0.04444136;
   W_g[9,16] := 0.07951424;
   W_g[9,17] := 0.00626671;
   W_g[9,18] := -0.06104251;
   W_g[9,19] := 0.04594292;
   W_g[9,20] := -0.02836513;
   W_g[9,21] := 0.0397499;
   W_g[9,22] := -0.02700124;
   W_g[9,23] := 0.02002714;
   W_g[9,24] := -0.5077276;
   W_g[9,25] := -0.2546269;
   W_g[9,26] := -0.03511217;
   W_g[9,27] := 0.04529352;
   W_g[9,28] := 0.04820129;
   W_g[9,29] := 0.09988645;
   W_g[9,30] := -0.01425081;
   W_g[9,31] := -0.01030078;
   W_g[9,32] := -0.01629252;
   W_g[9,33] := -0.00994037;
   W_g[9,34] := -0.5942311;
   W_g[9,35] := 0.03158842;
   W_g[9,36] := -0.08265782;
   W_g[9,37] := -0.0352644;
   W_g[9,38] := -0.00322891;
   W_g[9,39] := -0.00800959;
   W_g[10,0] := -0.03213325;
   W_g[10,1] := -0.00863164;
   W_g[10,2] := -0.03062097;
   W_g[10,3] := 0.0125538;
   W_g[10,4] := 0.1017359;
   W_g[10,5] := -0.04505892;
   W_g[10,6] := -0.00103756;
   W_g[10,7] := 0.01735601;
   W_g[10,8] := 0.01301922;
   W_g[10,9] := 0.0136564;
   W_g[10,10] := 0.00548952;
   W_g[10,11] := -0.00245858;
   W_g[10,12] := 0.00857112;
   W_g[10,13] := 0.1074988;
   W_g[10,14] := -0.1275509;
   W_g[10,15] := -0.03629598;
   W_g[10,16] := -0.01334849;
   W_g[10,17] := 0.1290663;
   W_g[10,18] := -0.01503343;
   W_g[10,19] := 0.01173486;
   W_g[10,20] := 0.06222534;
   W_g[10,21] := 0.05678142;
   W_g[10,22] := -0.02349397;
   W_g[10,23] := 0.06754656;
   W_g[10,24] := 0.1779617;
   W_g[10,25] := 0.1916296;
   W_g[10,26] := -0.02255434;
   W_g[10,27] := 0.1007323;
   W_g[10,28] := 0.1328024;
   W_g[10,29] := -0.01282987;
   W_g[10,30] := -0.01621767;
   W_g[10,31] := -0.0140665;
   W_g[10,32] := -0.00099214;
   W_g[10,33] := -0.00035058;
   W_g[10,34] := 0.1452188;
   W_g[10,35] := 0.02793738;
   W_g[10,36] := -0.07625148;
   W_g[10,37] := -0.00763791;
   W_g[10,38] := 0.00534324;
   W_g[10,39] := -0.3312542;
   W_g[11,0] := -0.1137508;
   W_g[11,1] := 0.05398307;
   W_g[11,2] := -0.1207509;
   W_g[11,3] := 0.04525032;
   W_g[11,4] := 0.08992387;
   W_g[11,5] := 0.01991016;
   W_g[11,6] := 0.2249754;
   W_g[11,7] := 0.04191377;
   W_g[11,8] := 0.04533296;
   W_g[11,9] := 0.0449999;
   W_g[11,10] := -0.1099455;
   W_g[11,11] := 0.00437518;
   W_g[11,12] := -0.00140931;
   W_g[11,13] := 0.04130397;
   W_g[11,14] := 0.053694;
   W_g[11,15] := -0.00366092;
   W_g[11,16] := -0.07105832;
   W_g[11,17] := -0.07482163;
   W_g[11,18] := -0.07100122;
   W_g[11,19] := 0.01718117;
   W_g[11,20] := -0.1375782;
   W_g[11,21] := 0.113075;
   W_g[11,22] := 0.054169;
   W_g[11,23] := 0.02884634;
   W_g[11,24] := 0.5307817;
   W_g[11,25] := 0.3570411;
   W_g[11,26] := 0.03378;
   W_g[11,27] := 0.1037555;
   W_g[11,28] := 0.2505002;
   W_g[11,29] := -0.1244629;
   W_g[11,30] := 0.0558193;
   W_g[11,31] := 0.05851344;
   W_g[11,32] := 0.07730477;
   W_g[11,33] := 0.09541148;
   W_g[11,34] := 0.1203315;
   W_g[11,35] := 0.1210543;
   W_g[11,36] := -0.1949756;
   W_g[11,37] := 0.0137196;
   W_g[11,38] := 0.08832928;
   W_g[11,39] := 0.08146589;
   W_g[12,0] := -0.02631861;
   W_g[12,1] := 0.04126604;
   W_g[12,2] := -0.02663527;
   W_g[12,3] := -0.02984582;
   W_g[12,4] := -0.02636349;
   W_g[12,5] := 0.07986053;
   W_g[12,6] := -0.01390989;
   W_g[12,7] := -0.00909171;
   W_g[12,8] := -0.01941176;
   W_g[12,9] := -0.02868326;
   W_g[12,10] := 0.03089914;
   W_g[12,11] := 0.00787742;
   W_g[12,12] := -0.00904082;
   W_g[12,13] := -0.0291048;
   W_g[12,14] := 0.1083951;
   W_g[12,15] := 0.01380038;
   W_g[12,16] := 0.06520407;
   W_g[12,17] := -0.04494612;
   W_g[12,18] := -0.0019409;
   W_g[12,19] := -0.0150968;
   W_g[12,20] := 0.08029543;
   W_g[12,21] := 0.02437602;
   W_g[12,22] := -0.07042312;
   W_g[12,23] := -0.04948704;
   W_g[12,24] := -0.8303994;
   W_g[12,25] := -0.5589937;
   W_g[12,26] := -0.04566456;
   W_g[12,27] := 0.0018911;
   W_g[12,28] := -0.02951618;
   W_g[12,29] := -0.05513477;
   W_g[12,30] := -0.04795056;
   W_g[12,31] := -0.0368838;
   W_g[12,32] := -0.03588131;
   W_g[12,33] := 0.00737297;
   W_g[12,34] := 0.0499457;
   W_g[12,35] := -0.01839683;
   W_g[12,36] := -0.4987357;
   W_g[12,37] := -0.07791845;
   W_g[12,38] := -0.1047491;
   W_g[12,39] := 0.00553967;
   W_g[13,0] := -0.0268404;
   W_g[13,1] := -0.088905;
   W_g[13,2] := -0.02790045;
   W_g[13,3] := 0.08189317;
   W_g[13,4] := -0.1255152;
   W_g[13,5] := -0.05772218;
   W_g[13,6] := 0.09080454;
   W_g[13,7] := 0.08241173;
   W_g[13,8] := 0.07553043;
   W_g[13,9] := 0.08949121;
   W_g[13,10] := -0.02704351;
   W_g[13,11] := 0.00487661;
   W_g[13,12] := 0.02095871;
   W_g[13,13] := 0.06879441;
   W_g[13,14] := 0.00018557;
   W_g[13,15] := 0.01617457;
   W_g[13,16] := 0.2304675;
   W_g[13,17] := 0.08005539;
   W_g[13,18] := -0.06847396;
   W_g[13,19] := 0.02106568;
   W_g[13,20] := -0.08102658;
   W_g[13,21] := -0.03850572;
   W_g[13,22] := 0.00878646;
   W_g[13,23] := 0.1475209;
   W_g[13,24] := 0.1967756;
   W_g[13,25] := -0.00969006;
   W_g[13,26] := 0.04820746;
   W_g[13,27] := -0.06298333;
   W_g[13,28] := -0.06368192;
   W_g[13,29] := 0.01809042;
   W_g[13,30] := 0.01814866;
   W_g[13,31] := 0.00847225;
   W_g[13,32] := 0.00546922;
   W_g[13,33] := -0.01145526;
   W_g[13,34] := 0.1381362;
   W_g[13,35] := 0.01473064;
   W_g[13,36] := -0.050091;
   W_g[13,37] := -0.01566363;
   W_g[13,38] := 0.05946118;
   W_g[13,39] := 0.00826691;
   W_g[14,0] := 0.02104861;
   W_g[14,1] := 0.02198478;
   W_g[14,2] := 0.0111862;
   W_g[14,3] := -0.06436396;
   W_g[14,4] := 0.00489476;
   W_g[14,5] := 0.09250024;
   W_g[14,6] := -0.03399736;
   W_g[14,7] := -0.0496763;
   W_g[14,8] := -0.05370576;
   W_g[14,9] := -0.05536002;
   W_g[14,10] := 0.01229766;
   W_g[14,11] := -0.01784988;
   W_g[14,12] := -0.03607991;
   W_g[14,13] := 0.1900748;
   W_g[14,14] := 0.08048796;
   W_g[14,15] := -0.0089345;
   W_g[14,16] := 0.01208448;
   W_g[14,17] := -0.06566814;
   W_g[14,18] := -0.2211387;
   W_g[14,19] := -0.04166633;
   W_g[14,20] := 0.07567322;
   W_g[14,21] := -0.00166608;
   W_g[14,22] := -0.01256561;
   W_g[14,23] := 0.1539435;
   W_g[14,24] := 0.03526039;
   W_g[14,25] := 0.4811959;
   W_g[14,26] := 0.01489335;
   W_g[14,27] := 0.0317387;
   W_g[14,28] := 0.01991428;
   W_g[14,29] := 0.03107417;
   W_g[14,30] := -0.00682632;
   W_g[14,31] := 0.00660902;
   W_g[14,32] := 0.00283587;
   W_g[14,33] := -0.00859028;
   W_g[14,34] := -0.02930867;
   W_g[14,35] := 0.03631073;
   W_g[14,36] := 0.00467363;
   W_g[14,37] := 0.02703222;
   W_g[14,38] := -0.04237745;
   W_g[14,39] := 0.01309555;
   W_g[15,0] := 0.08495549;
   W_g[15,1] := -0.2072809;
   W_g[15,2] := 0.08629236;
   W_g[15,3] := -0.06330224;
   W_g[15,4] := 0.1923753;
   W_g[15,5] := 0.00801008;
   W_g[15,6] := -0.104994;
   W_g[15,7] := -0.05814644;
   W_g[15,8] := -0.06757385;
   W_g[15,9] := -0.0590176;
   W_g[15,10] := -0.00683508;
   W_g[15,11] := -0.00540838;
   W_g[15,12] := -0.02551957;
   W_g[15,13] := -0.01507952;
   W_g[15,14] := 0.00483655;
   W_g[15,15] := 0.01358667;
   W_g[15,16] := 0.2541837;
   W_g[15,17] := -0.01636837;
   W_g[15,18] := 0.01947031;
   W_g[15,19] := -0.03640394;
   W_g[15,20] := 0.2146612;
   W_g[15,21] := 0.1069127;
   W_g[15,22] := 0.03332973;
   W_g[15,23] := -0.06589723;
   W_g[15,24] := 0.1503799;
   W_g[15,25] := 0.03056319;
   W_g[15,26] := -0.08210966;
   W_g[15,27] := 0.1496714;
   W_g[15,28] := 0.09097399;
   W_g[15,29] := -0.04645663;
   W_g[15,30] := 0.04627259;
   W_g[15,31] := 0.00594573;
   W_g[15,32] := 0.05130993;
   W_g[15,33] := 0.05626767;
   W_g[15,34] := -0.00315162;
   W_g[15,35] := 0.04370028;
   W_g[15,36] := -0.06999733;
   W_g[15,37] := 0.01681984;
   W_g[15,38] := 0.0727107;
   W_g[15,39] := 0.01082875;
   W_o[0,0] := -0.1923357;
   W_o[0,1] := 0.1622824;
   W_o[0,2] := 0.03764162;
   W_o[0,3] := -0.00444271;
   W_o[0,4] := 0.0897337;
   W_o[0,5] := 0.05718408;
   W_o[0,6] := -0.2313943;
   W_o[0,7] := 0.1578357;
   W_o[0,8] := -0.1582883;
   W_o[0,9] := 0.1973625;
   W_o[0,10] := -0.3052712;
   W_o[0,11] := -0.2301492;
   W_o[0,12] := 0.209668;
   W_o[0,13] := -0.1742153;
   W_o[0,14] := -0.2678694;
   W_o[0,15] := -0.01321167;
   W_o[0,16] := -0.01970488;
   W_o[0,17] := -0.2028062;
   W_o[0,18] := 0.4272551;
   W_o[0,19] := -0.06582518;
   W_o[0,20] := -0.03046696;
   W_o[0,21] := 0.5501582;
   W_o[0,22] := 0.4423466;
   W_o[0,23] := -0.3345911;
   W_o[0,24] := 1.265247;
   W_o[0,25] := 1.416652;
   W_o[0,26] := -0.3267373;
   W_o[0,27] := -0.1832035;
   W_o[0,28] := 0.01126313;
   W_o[0,29] := -0.2838583;
   W_o[0,30] := 0.2609881;
   W_o[0,31] := 0.04669111;
   W_o[0,32] := 0.1043487;
   W_o[0,33] := 0.05575988;
   W_o[0,34] := 1.332353;
   W_o[0,35] := -0.06145113;
   W_o[0,36] := -0.0334513;
   W_o[0,37] := -0.2221547;
   W_o[0,38] := 0.00487359;
   W_o[0,39] := -0.03890218;
   W_o[1,0] := 0.7437804;
   W_o[1,1] := -0.0500013;
   W_o[1,2] := 0.1212982;
   W_o[1,3] := 0.1032013;
   W_o[1,4] := 0.1199842;
   W_o[1,5] := -0.1907221;
   W_o[1,6] := 0.2100161;
   W_o[1,7] := 0.1133247;
   W_o[1,8] := 0.3588262;
   W_o[1,9] := 0.3857575;
   W_o[1,10] := -0.4587842;
   W_o[1,11] := -0.1574819;
   W_o[1,12] := 0.2066407;
   W_o[1,13] := 0.1230617;
   W_o[1,14] := -0.203037;
   W_o[1,15] := 0.03768912;
   W_o[1,16] := -0.05619529;
   W_o[1,17] := -0.09439399;
   W_o[1,18] := 0.2707254;
   W_o[1,19] := 0.3822214;
   W_o[1,20] := -0.2934351;
   W_o[1,21] := 0.5161377;
   W_o[1,22] := 0.1759103;
   W_o[1,23] := 0.1837359;
   W_o[1,24] := -0.03005522;
   W_o[1,25] := 0.00781888;
   W_o[1,26] := -0.1068488;
   W_o[1,27] := -0.07173182;
   W_o[1,28] := 0.2014527;
   W_o[1,29] := 0.1306461;
   W_o[1,30] := -0.01024106;
   W_o[1,31] := -0.0716324;
   W_o[1,32] := 0.05804014;
   W_o[1,33] := 0.2721744;
   W_o[1,34] := 0.06194695;
   W_o[1,35] := -0.304073;
   W_o[1,36] := 0.1530892;
   W_o[1,37] := -0.07396729;
   W_o[1,38] := 0.08739793;
   W_o[1,39] := 0.3265531;
   W_o[2,0] := -0.03605163;
   W_o[2,1] := 0.07661975;
   W_o[2,2] := 0.1369504;
   W_o[2,3] := 0.09188601;
   W_o[2,4] := 0.03664814;
   W_o[2,5] := -0.02675835;
   W_o[2,6] := -0.01984608;
   W_o[2,7] := -0.1901468;
   W_o[2,8] := -0.02938575;
   W_o[2,9] := 0.1836661;
   W_o[2,10] := -0.1862541;
   W_o[2,11] := 0.06671655;
   W_o[2,12] := 0.3190728;
   W_o[2,13] := -0.01547686;
   W_o[2,14] := -0.05195596;
   W_o[2,15] := 0.03504787;
   W_o[2,16] := 0.3541903;
   W_o[2,17] := 0.02718459;
   W_o[2,18] := -0.2491126;
   W_o[2,19] := -0.8667619;
   W_o[2,20] := -0.1266757;
   W_o[2,21] := 0.02015731;
   W_o[2,22] := -0.02294585;
   W_o[2,23] := -0.01648583;
   W_o[2,24] := -0.1919154;
   W_o[2,25] := 0.00051678;
   W_o[2,26] := 0.06543333;
   W_o[2,27] := 0.1037415;
   W_o[2,28] := -0.0450457;
   W_o[2,29] := 0.215062;
   W_o[2,30] := 0.02658869;
   W_o[2,31] := -0.1369152;
   W_o[2,32] := 0.01719045;
   W_o[2,33] := 0.218743;
   W_o[2,34] := -0.07076459;
   W_o[2,35] := -0.0740788;
   W_o[2,36] := -0.08052358;
   W_o[2,37] := -0.2012888;
   W_o[2,38] := -0.3849033;
   W_o[2,39] := 0.6891636;
   W_o[3,0] := -0.06302688;
   W_o[3,1] := 0.2002212;
   W_o[3,2] := 0.0159587;
   W_o[3,3] := -0.0018361;
   W_o[3,4] := -0.8591735;
   W_o[3,5] := 0.1731812;
   W_o[3,6] := 0.2409841;
   W_o[3,7] := 0.2596082;
   W_o[3,8] := -0.00940404;
   W_o[3,9] := 0.06814823;
   W_o[3,10] := -0.01664601;
   W_o[3,11] := 0.148778;
   W_o[3,12] := -0.09583785;
   W_o[3,13] := -0.2798349;
   W_o[3,14] := 0.1443422;
   W_o[3,15] := 0.00555357;
   W_o[3,16] := -0.02839783;
   W_o[3,17] := 0.09947813;
   W_o[3,18] := 0.4643263;
   W_o[3,19] := 0.0636435;
   W_o[3,20] := -0.08531965;
   W_o[3,21] := 1.165775;
   W_o[3,22] := 0.3448276;
   W_o[3,23] := -0.117277;
   W_o[3,24] := 1.352477;
   W_o[3,25] := 1.178241;
   W_o[3,26] := -0.4892529;
   W_o[3,27] := -0.7737502;
   W_o[3,28] := 0.2264518;
   W_o[3,29] := 0.00574818;
   W_o[3,30] := 0.2461463;
   W_o[3,31] := 0.1052826;
   W_o[3,32] := 0.00088265;
   W_o[3,33] := 0.1049805;
   W_o[3,34] := 1.18573;
   W_o[3,35] := 0.1909419;
   W_o[3,36] := -0.00811989;
   W_o[3,37] := 0.09236411;
   W_o[3,38] := 0.1108437;
   W_o[3,39] := 0.9237891;
   W_o[4,0] := -0.1855668;
   W_o[4,1] := -0.06182796;
   W_o[4,2] := 0.1497869;
   W_o[4,3] := -0.02874054;
   W_o[4,4] := -0.2372189;
   W_o[4,5] := -0.02661614;
   W_o[4,6] := 0.04865195;
   W_o[4,7] := -0.2595509;
   W_o[4,8] := 0.5146528;
   W_o[4,9] := -0.2822051;
   W_o[4,10] := 0.01177313;
   W_o[4,11] := -0.4989094;
   W_o[4,12] := -0.8648744;
   W_o[4,13] := -0.04488994;
   W_o[4,14] := -0.0542339;
   W_o[4,15] := -0.5589076;
   W_o[4,16] := -0.145594;
   W_o[4,17] := 0.02167914;
   W_o[4,18] := 1.006644;
   W_o[4,19] := -0.2599575;
   W_o[4,20] := 0.00703312;
   W_o[4,21] := -0.2283233;
   W_o[4,22] := 0.00192229;
   W_o[4,23] := -0.01435418;
   W_o[4,24] := 0.04472705;
   W_o[4,25] := 0.2338529;
   W_o[4,26] := -0.1127145;
   W_o[4,27] := 0.08130027;
   W_o[4,28] := 0.4603895;
   W_o[4,29] := 0.1379606;
   W_o[4,30] := 0.1812189;
   W_o[4,31] := -0.3901244;
   W_o[4,32] := -0.0703788;
   W_o[4,33] := 0.2888122;
   W_o[4,34] := 0.4034505;
   W_o[4,35] := 0.0328819;
   W_o[4,36] := -0.09105004;
   W_o[4,37] := 0.09711539;
   W_o[4,38] := -0.1910721;
   W_o[4,39] := -0.01934181;
   W_o[5,0] := -0.6595194;
   W_o[5,1] := 0.3772199;
   W_o[5,2] := 0.00501744;
   W_o[5,3] := 0.532542;
   W_o[5,4] := 0.2366183;
   W_o[5,5] := 1.09201;
   W_o[5,6] := 0.9502543;
   W_o[5,7] := 0.2582511;
   W_o[5,8] := -0.4691281;
   W_o[5,9] := 0.3928114;
   W_o[5,10] := 1.11464;
   W_o[5,11] := -0.7781826;
   W_o[5,12] := -0.6074764;
   W_o[5,13] := 0.16801;
   W_o[5,14] := -0.1086531;
   W_o[5,15] := -0.6841738;
   W_o[5,16] := -0.3678641;
   W_o[5,17] := -0.2172338;
   W_o[5,18] := 0.3863191;
   W_o[5,19] := -0.4950597;
   W_o[5,20] := -0.5119882;
   W_o[5,21] := -0.1780492;
   W_o[5,22] := 0.1544936;
   W_o[5,23] := 0.1383117;
   W_o[5,24] := 1.004889;
   W_o[5,25] := 1.139415;
   W_o[5,26] := -0.3015366;
   W_o[5,27] := -0.04238907;
   W_o[5,28] := -0.3108428;
   W_o[5,29] := 0.3969988;
   W_o[5,30] := 0.01171695;
   W_o[5,31] := -0.3139689;
   W_o[5,32] := -0.3243381;
   W_o[5,33] := -0.414901;
   W_o[5,34] := 0.2215569;
   W_o[5,35] := -0.133694;
   W_o[5,36] := 0.02332771;
   W_o[5,37] := -0.1487403;
   W_o[5,38] := 0.1979396;
   W_o[5,39] := -0.2030152;
   W_o[6,0] := -0.04529256;
   W_o[6,1] := 0.2150283;
   W_o[6,2] := 0.09295318;
   W_o[6,3] := -0.0767066;
   W_o[6,4] := -0.1236452;
   W_o[6,5] := 0.3573766;
   W_o[6,6] := -0.2646887;
   W_o[6,7] := 0.2834802;
   W_o[6,8] := -0.04882327;
   W_o[6,9] := 0.8413;
   W_o[6,10] := 1.089968;
   W_o[6,11] := -0.06981075;
   W_o[6,12] := 0.05921048;
   W_o[6,13] := -0.5099319;
   W_o[6,14] := 0.04131682;
   W_o[6,15] := 0.09513918;
   W_o[6,16] := 0.08072844;
   W_o[6,17] := 0.02096614;
   W_o[6,18] := 0.1683812;
   W_o[6,19] := 0.1104724;
   W_o[6,20] := -0.3392214;
   W_o[6,21] := -0.09979945;
   W_o[6,22] := 0.1501902;
   W_o[6,23] := -0.06504018;
   W_o[6,24] := 1.949389;
   W_o[6,25] := 1.979982;
   W_o[6,26] := 0.02307883;
   W_o[6,27] := 0.2684888;
   W_o[6,28] := 0.09674384;
   W_o[6,29] := 0.2116341;
   W_o[6,30] := 0.1413678;
   W_o[6,31] := -0.0124489;
   W_o[6,32] := -0.04519035;
   W_o[6,33] := -0.1396772;
   W_o[6,34] := 0.4939206;
   W_o[6,35] := -0.2130735;
   W_o[6,36] := 0.06053885;
   W_o[6,37] := 0.0587407;
   W_o[6,38] := 0.429702;
   W_o[6,39] := -0.1062183;
   W_o[7,0] := 0.1648133;
   W_o[7,1] := -0.09838933;
   W_o[7,2] := -0.0939215;
   W_o[7,3] := -0.1272545;
   W_o[7,4] := -0.2333547;
   W_o[7,5] := 0.05955706;
   W_o[7,6] := 0.2717095;
   W_o[7,7] := 0.1100897;
   W_o[7,8] := 0.1809682;
   W_o[7,9] := 0.01596895;
   W_o[7,10] := 0.1498611;
   W_o[7,11] := -0.3100757;
   W_o[7,12] := 0.5308929;
   W_o[7,13] := -0.07378945;
   W_o[7,14] := -0.2509805;
   W_o[7,15] := 0.2649329;
   W_o[7,16] := -0.1476106;
   W_o[7,17] := -0.2392291;
   W_o[7,18] := 0.4080176;
   W_o[7,19] := -0.1504776;
   W_o[7,20] := -0.1111432;
   W_o[7,21] := 0.1132136;
   W_o[7,22] := 0.464526;
   W_o[7,23] := -0.1314203;
   W_o[7,24] := 0.8524858;
   W_o[7,25] := 0.9319458;
   W_o[7,26] := 0.1910378;
   W_o[7,27] := -0.04179411;
   W_o[7,28] := 0.1727818;
   W_o[7,29] := -0.3418947;
   W_o[7,30] := 0.4730469;
   W_o[7,31] := 0.08789608;
   W_o[7,32] := 0.2170709;
   W_o[7,33] := -0.03279238;
   W_o[7,34] := 0.6582685;
   W_o[7,35] := 0.08038806;
   W_o[7,36] := 0.04812925;
   W_o[7,37] := 0.4378351;
   W_o[7,38] := -0.06570955;
   W_o[7,39] := -1.681702;
   W_o[8,0] := 0.2838559;
   W_o[8,1] := -0.1376109;
   W_o[8,2] := -0.00303996;
   W_o[8,3] := -0.1514946;
   W_o[8,4] := -0.05367951;
   W_o[8,5] := 0.3758456;
   W_o[8,6] := 0.02626968;
   W_o[8,7] := -0.1422179;
   W_o[8,8] := 0.00944922;
   W_o[8,9] := -0.2079319;
   W_o[8,10] := -0.2131251;
   W_o[8,11] := -1.025984;
   W_o[8,12] := -0.3985277;
   W_o[8,13] := -0.0818603;
   W_o[8,14] := -0.1052002;
   W_o[8,15] := -1.120577;
   W_o[8,16] := 0.05219958;
   W_o[8,17] := 0.7909105;
   W_o[8,18] := 0.3779635;
   W_o[8,19] := 0.16329;
   W_o[8,20] := -0.06752818;
   W_o[8,21] := 0.2244961;
   W_o[8,22] := -0.133298;
   W_o[8,23] := -0.5498607;
   W_o[8,24] := 0.210675;
   W_o[8,25] := 0.4249826;
   W_o[8,26] := 0.3085507;
   W_o[8,27] := 0.00327513;
   W_o[8,28] := -0.1328674;
   W_o[8,29] := 0.2423343;
   W_o[8,30] := -0.2916745;
   W_o[8,31] := 0.1113145;
   W_o[8,32] := 0.235408;
   W_o[8,33] := 0.2593887;
   W_o[8,34] := 0.2619374;
   W_o[8,35] := 0.09260385;
   W_o[8,36] := -0.07284077;
